LIN {X 0,Y 573.238,Z 329.704,A -85,B 0,C 180,E1 -2317.662,E2 -2317.662} C_VEL
LIN {X 0,Y 573.282,Z 329.698,A -85,B 0,C 180,E1 -2320.728,E2 -2320.728} C_VEL
LIN {X 0,Y 573.255,Z 329.702,A -85,B 0,C 180,E1 -2323.622,E2 -2323.622} C_VEL
LIN {X 0,Y 573.278,Z 329.701,A -85,B 0,C 180,E1 -2325.807,E2 -2325.807} C_VEL
LIN {X 0,Y 573.267,Z 329.702,A -85,B 0,C 180,E1 -2328.745,E2 -2328.745} C_VEL
LIN {X 0,Y 573.287,Z 329.698,A -85,B 0,C 180,E1 -2331.541,E2 -2331.541} C_VEL
LIN {X 0,Y 573.291,Z 329.697,A -85,B 0,C 180,E1 -2334.372,E2 -2334.372} C_VEL
LIN {X 0,Y 573.311,Z 329.696,A -85,B 0,C 180,E1 -2337.893,E2 -2337.893} C_VEL
LIN {X 0,Y 573.336,Z 329.691,A -85,B 0,C 180,E1 -2340.702,E2 -2340.702} C_VEL
LIN {X 0,Y 573.239,Z 329.703,A -85,B 0,C 180,E1 -2343.515,E2 -2343.515} C_VEL
LIN {X 0,Y 573.297,Z 329.699,A -85,B 0,C 180,E1 -2345.628,E2 -2345.628} C_VEL
LIN {X 0,Y 573.292,Z 329.697,A -85,B 0,C 180,E1 -2348.459,E2 -2348.459} C_VEL
LIN {X 0,Y 573.276,Z 329.697,A -85,B 0,C 180,E1 -2351.312,E2 -2351.312} C_VEL
LIN {X 0,Y 573.285,Z 329.696,A -85,B 0,C 180,E1 -2354.424,E2 -2354.424} C_VEL
LIN {X 0,Y 573.264,Z 329.701,A -85,B 0,C 180,E1 -2357.112,E2 -2357.112} C_VEL
LIN {X 0,Y 573.255,Z 329.699,A -85,B 0,C 180,E1 -2360.077,E2 -2360.077} C_VEL
LIN {X 0,Y 573.238,Z 329.704,A -85,B 0,C 180,E1 -2363.099,E2 -2363.099} C_VEL
LIN {X 0,Y 573.252,Z 329.701,A -85,B 0,C 180,E1 -2364.385,E2 -2364.385} C_VEL
LIN {X 0,Y 572.628,Z 329.781,A -85,B 0,C 180,E1 -2364.971,E2 -2364.971} C_VEL
LIN {X 0,Y 569.787,Z 330.139,A -85,B 0,C 180,E1 -2365.922,E2 -2365.922} C_VEL
LIN {X 0,Y 567.354,Z 330.442,A -85,B 0,C 180,E1 -2366.688,E2 -2366.688} C_VEL
LIN {X 0,Y 566.298,Z 330.571,A -85,B 0,C 180,E1 -2367.279,E2 -2367.279} C_VEL
LIN {X 0,Y 566.207,Z 330.58,A -85,B 0,C 180,E1 -2367.479,E2 -2367.479} C_VEL
LIN {X 0,Y 566.205,Z 330.58,A -85,B 0,C 180,E1 -2369.769,E2 -2369.769} C_VEL
LIN {X 0,Y 566.207,Z 330.578,A -85,B 0,C 180,E1 -2372.43,E2 -2372.43} C_VEL
LIN {X 0,Y 566.206,Z 330.584,A -85,B 0,C 180,E1 -2374.993,E2 -2374.993} C_VEL
LIN {X 0,Y 566.2,Z 330.581,A -85,B 0,C 180,E1 -2377.461,E2 -2377.461} C_VEL
LIN {X 0,Y 566.222,Z 330.578,A -85,B 0,C 180,E1 -2380.198,E2 -2380.198} C_VEL
LIN {X 0,Y 566.204,Z 330.58,A -85,B 0,C 180,E1 -2383.054,E2 -2383.054} C_VEL
LIN {X 0,Y 566.202,Z 330.581,A -85,B 0,C 180,E1 -2386.049,E2 -2386.049} C_VEL
LIN {X 0,Y 566.132,Z 330.595,A -85,B 0,C 180,E1 -2388.856,E2 -2388.856} C_VEL
LIN {X 0,Y 566.084,Z 331.003,A -85,B 0,C 180,E1 -2389.79,E2 -2389.79} C_VEL
LIN {X 0,Y 566.074,Z 333.817,A -85,B 0,C 180,E1 -2392.616,E2 -2392.616} C_VEL
LIN {X 0,Y 566.042,Z 336.324,A -85,B 0,C 180,E1 -2395.17,E2 -2395.17} C_VEL
LIN {X 0,Y 566.028,Z 338.882,A -85,B 0,C 180,E1 -2397.73,E2 -2397.73} C_VEL
LIN {X 0,Y 566.001,Z 341.587,A -85,B 0,C 180,E1 -2400.364,E2 -2400.364} C_VEL
LIN {X 0,Y 565.931,Z 344.797,A -85,B 0,C 180,E1 -2403.444,E2 -2403.444} C_VEL
LIN {X 0,Y 565.906,Z 347.412,A -85,B 0,C 180,E1 -2405.806,E2 -2405.806} C_VEL
LIN {X 0,Y 565.904,Z 351.128,A -85,B 0,C 180,E1 -2408.89,E2 -2408.89} C_VEL
LIN {X 0,Y 565.866,Z 354.845,A -85,B 0,C 180,E1 -2411.911,E2 -2411.911} C_VEL
LIN {X 0,Y 565.878,Z 355.244,A -85,B 0,C 180,E1 -2412.232,E2 -2412.232} C_VEL
LIN {X 0,Y 567.937,Z 363.992,A -85,B 0,C 180,E1 -2412.448,E2 -2412.448} C_VEL
LIN {X 0,Y 567.807,Z 378.874,A -85,B 0,C 180,E1 -2412.799,E2 -2412.799} C_VEL
LIN {X 0,Y 567.62,Z 393.572,A -85,B 0,C 180,E1 -2413.29,E2 -2413.29} C_VEL
LIN {X 0,Y 567.404,Z 407.73,A -85,B 0,C 180,E1 -2413.91,E2 -2413.91} C_VEL
LIN {X 0,Y 567.144,Z 421.039,A -85,B 0,C 180,E1 -2414.64,E2 -2414.64} C_VEL
LIN {X 0,Y 566.919,Z 433.971,A -85,B 0,C 180,E1 -2415.507,E2 -2415.507} C_VEL
LIN {X 0,Y 566.651,Z 446.885,A -85,B 0,C 180,E1 -2416.552,E2 -2416.552} C_VEL
LIN {X 0,Y 566.463,Z 458.082,A -85,B 0,C 180,E1 -2417.642,E2 -2417.642} C_VEL
LIN {X 0,Y 566.264,Z 468.177,A -85,B 0,C 180,E1 -2418.809,E2 -2418.809} C_VEL
LIN {X 0,Y 566.133,Z 478.002,A -85,B 0,C 180,E1 -2420.172,E2 -2420.172} C_VEL
LIN {X 0,Y 566.064,Z 485.494,A -85,B 0,C 180,E1 -2421.431,E2 -2421.431} C_VEL
LIN {X 0,Y 565.976,Z 492.498,A -85,B 0,C 180,E1 -2422.867,E2 -2422.867} C_VEL
LIN {X 0,Y 565.982,Z 498.007,A -85,B 0,C 180,E1 -2424.299,E2 -2424.299} C_VEL
LIN {X 0,Y 565.913,Z 502.177,A -85,B 0,C 180,E1 -2425.726,E2 -2425.726} C_VEL
LIN {X 0,Y 565.872,Z 505.114,A -85,B 0,C 180,E1 -2427.152,E2 -2427.152} C_VEL
LIN {X 0,Y 565.842,Z 506.88,A -85,B 0,C 180,E1 -2428.576,E2 -2428.576} C_VEL
LIN {X 0,Y 565.837,Z 507.496,A -85,B 0,C 180,E1 -2430,E2 -2430} C_VEL
LIN {X 0,Y 565.844,Z 506.942,A -85,B 0,C 180,E1 -2431.423,E2 -2431.423} C_VEL
LIN {X 0,Y 565.874,Z 505.259,A -85,B 0,C 180,E1 -2432.847,E2 -2432.847} C_VEL
LIN {X 0,Y 565.913,Z 502.404,A -85,B 0,C 180,E1 -2434.273,E2 -2434.273} C_VEL
LIN {X 0,Y 565.975,Z 498.319,A -85,B 0,C 180,E1 -2435.701,E2 -2435.701} C_VEL
LIN {X 0,Y 565.975,Z 492.905,A -85,B 0,C 180,E1 -2437.133,E2 -2437.133} C_VEL
LIN {X 0,Y 566.061,Z 486.005,A -85,B 0,C 180,E1 -2438.568,E2 -2438.568} C_VEL
LIN {X 0,Y 566.177,Z 477.397,A -85,B 0,C 180,E1 -2440.008,E2 -2440.008} C_VEL
LIN {X 0,Y 566.25,Z 468.953,A -85,B 0,C 180,E1 -2441.183,E2 -2441.183} C_VEL
LIN {X 0,Y 566.436,Z 458.917,A -85,B 0,C 180,E1 -2442.358,E2 -2442.358} C_VEL
LIN {X 0,Y 566.668,Z 446.873,A -85,B 0,C 180,E1 -2443.538,E2 -2443.538} C_VEL
LIN {X 0,Y 566.871,Z 435.302,A -85,B 0,C 180,E1 -2444.484,E2 -2444.484} C_VEL
LIN {X 0,Y 567.148,Z 422.48,A -85,B 0,C 180,E1 -2445.359,E2 -2445.359} C_VEL
LIN {X 0,Y 567.374,Z 409.469,A -85,B 0,C 180,E1 -2446.09,E2 -2446.09} C_VEL
LIN {X 0,Y 567.587,Z 395.421,A -85,B 0,C 180,E1 -2446.725,E2 -2446.725} C_VEL
LIN {X 0,Y 567.79,Z 380.271,A -85,B 0,C 180,E1 -2447.249,E2 -2447.249} C_VEL
LIN {X 0,Y 567.911,Z 365.71,A -85,B 0,C 180,E1 -2447.608,E2 -2447.608} C_VEL
LIN {X 0,Y 567.553,Z 362.338,A -85,B 0,C 180,E1 -2447.688,E2 -2447.688} C_VEL
LIN {X 0,Y 565.868,Z 355.244,A -85,B 0,C 180,E1 -2447.858,E2 -2447.858} C_VEL
LIN {X 0,Y 565.88,Z 352.168,A -85,B 0,C 180,E1 -2450.349,E2 -2450.349} C_VEL
LIN {X 0,Y 565.895,Z 348.449,A -85,B 0,C 180,E1 -2453.416,E2 -2453.416} C_VEL
LIN {X 0,Y 565.942,Z 345.739,A -85,B 0,C 180,E1 -2455.762,E2 -2455.762} C_VEL
LIN {X 0,Y 565.96,Z 343.279,A -85,B 0,C 180,E1 -2458.156,E2 -2458.156} C_VEL
LIN {X 0,Y 566.006,Z 340.226,A -85,B 0,C 180,E1 -2461.045,E2 -2461.045} C_VEL
LIN {X 0,Y 566.049,Z 337.269,A -85,B 0,C 180,E1 -2463.967,E2 -2463.967} C_VEL
LIN {X 0,Y 566.046,Z 334.704,A -85,B 0,C 180,E1 -2466.581,E2 -2466.581} C_VEL
LIN {X 0,Y 566.062,Z 332.025,A -85,B 0,C 180,E1 -2469.286,E2 -2469.286} C_VEL
LIN {X 0,Y 566.078,Z 330.601,A -85,B 0,C 180,E1 -2470.77,E2 -2470.77} C_VEL
LIN {X 0,Y 566.205,Z 330.585,A -85,B 0,C 180,E1 -2473.053,E2 -2473.053} C_VEL
LIN {X 0,Y 566.198,Z 330.586,A -85,B 0,C 180,E1 -2476.048,E2 -2476.048} C_VEL
LIN {X 0,Y 566.208,Z 330.582,A -85,B 0,C 180,E1 -2478.863,E2 -2478.863} C_VEL
LIN {X 0,Y 566.19,Z 330.582,A -85,B 0,C 180,E1 -2481.637,E2 -2481.637} C_VEL
LIN {X 0,Y 566.212,Z 330.579,A -85,B 0,C 180,E1 -2484.311,E2 -2484.311} C_VEL
LIN {X 0,Y 566.219,Z 330.58,A -85,B 0,C 180,E1 -2486.898,E2 -2486.898} C_VEL
LIN {X 0,Y 566.193,Z 330.582,A -85,B 0,C 180,E1 -2489.408,E2 -2489.408} C_VEL
LIN {X 0,Y 566.227,Z 330.575,A -85,B 0,C 180,E1 -2491.858,E2 -2491.858} C_VEL
LIN {X 0,Y 566.225,Z 330.58,A -85,B 0,C 180,E1 -2494.251,E2 -2494.251} C_VEL
LIN {X 0,Y 566.191,Z 330.581,A -85,B 0,C 180,E1 -2496.713,E2 -2496.713} C_VEL
LIN {X 0,Y 566.213,Z 330.575,A -85,B 0,C 180,E1 -2499.663,E2 -2499.663} C_VEL
LIN {X 0,Y 566.203,Z 330.58,A -85,B 0,C 180,E1 -2502.668,E2 -2502.668} C_VEL
LIN {X 0,Y 566.233,Z 330.574,A -85,B 0,C 180,E1 -2505.627,E2 -2505.627} C_VEL
LIN {X 0,Y 566.233,Z 330.575,A -85,B 0,C 180,E1 -2508.675,E2 -2508.675} C_VEL
LIN {X 0,Y 566.233,Z 330.578,A -85,B 0,C 180,E1 -2511.434,E2 -2511.434} C_VEL
LIN {X 0,Y 566.263,Z 330.576,A -85,B 0,C 180,E1 -2514.302,E2 -2514.302} C_VEL
LIN {X 0,Y 566.277,Z 330.571,A -85,B 0,C 180,E1 -2517.866,E2 -2517.866} C_VEL
LIN {X 0,Y 566.303,Z 330.568,A -85,B 0,C 180,E1 -2520.711,E2 -2520.711} C_VEL
LIN {X 0,Y 566.276,Z 330.572,A -85,B 0,C 180,E1 -2522.845,E2 -2522.845} C_VEL
LIN {X 0,Y 566.259,Z 330.573,A -85,B 0,C 180,E1 -2525.698,E2 -2525.698} C_VEL
LIN {X 0,Y 566.228,Z 330.577,A -85,B 0,C 180,E1 -2528.566,E2 -2528.566} C_VEL
LIN {X 0,Y 566.25,Z 330.574,A -85,B 0,C 180,E1 -2531.454,E2 -2531.454} C_VEL
LIN {X 0,Y 566.233,Z 330.576,A -85,B 0,C 180,E1 -2534.507,E2 -2534.507} C_VEL
LIN {X 0,Y 566.199,Z 330.582,A -85,B 0,C 180,E1 -2537.332,E2 -2537.332} C_VEL
LIN {X 0,Y 566.212,Z 330.58,A -85,B 0,C 180,E1 -2540.337,E2 -2540.337} C_VEL
LIN {X 0,Y 566.188,Z 330.584,A -85,B 0,C 180,E1 -2543.404,E2 -2543.404} C_VEL
LIN {X 0,Y 566.212,Z 330.581,A -85,B 0,C 180,E1 -2545.749,E2 -2545.749} C_VEL
LIN {X 0,Y 566.2,Z 330.581,A -85,B 0,C 180,E1 -2548.202,E2 -2548.202} C_VEL
LIN {X 0,Y 566.193,Z 330.586,A -85,B 0,C 180,E1 -2550.592,E2 -2550.592} C_VEL
LIN {X 0,Y 566.227,Z 330.578,A -85,B 0,C 180,E1 -2553.102,E2 -2553.102} C_VEL
LIN {X 0,Y 566.211,Z 330.581,A -85,B 0,C 180,E1 -2555.689,E2 -2555.689} C_VEL
LIN {X 0,Y 566.216,Z 330.581,A -85,B 0,C 180,E1 -2558.559,E2 -2558.559} C_VEL
LIN {X 0,Y 566.211,Z 330.583,A -85,B 0,C 180,E1 -2561.136,E2 -2561.136} C_VEL
LIN {X 0,Y 566.195,Z 330.584,A -85,B 0,C 180,E1 -2564.036,E2 -2564.036} C_VEL
LIN {X 0,Y 566.24,Z 330.749,A -85,B 0,C 180,E1 -2567.079,E2 -2567.079} C_VEL
LIN {X 0,Y 566.797,Z 335.443,A -85,B 0,C 180,E1 -2569.145,E2 -2569.145} C_VEL
LIN {X 0,Y 566.637,Z 342.907,A -85,B 0,C 180,E1 -2572.125,E2 -2572.125} C_VEL
LIN {X 0,Y 566.573,Z 348.853,A -85,B 0,C 180,E1 -2574.338,E2 -2574.338} C_VEL
LIN {X 0,Y 566.495,Z 356.024,A -85,B 0,C 180,E1 -2576.916,E2 -2576.916} C_VEL
LIN {X 0,Y 566.454,Z 363.225,A -85,B 0,C 180,E1 -2579.424,E2 -2579.424} C_VEL
LIN {X 0,Y 566.367,Z 371.685,A -85,B 0,C 180,E1 -2582.269,E2 -2582.269} C_VEL
LIN {X 0,Y 566.318,Z 379.997,A -85,B 0,C 180,E1 -2585.043,E2 -2585.043} C_VEL
LIN {X 0,Y 566.207,Z 389.338,A -85,B 0,C 180,E1 -2588.138,E2 -2588.138} C_VEL
LIN {X 0,Y 566.13,Z 398.678,A -85,B 0,C 180,E1 -2591.17,E2 -2591.17} C_VEL
LIN {X 0,Y 566.103,Z 401.758,A -85,B 0,C 180,E1 -2592.152,E2 -2592.152} C_VEL
LIN {X 0,Y 567.951,Z 409.837,A -85,B 0,C 180,E1 -2592.33,E2 -2592.33} C_VEL
LIN {X 0,Y 567.836,Z 425.005,A -85,B 0,C 180,E1 -2592.65,E2 -2592.65} C_VEL
LIN {X 0,Y 567.714,Z 439.216,A -85,B 0,C 180,E1 -2593.087,E2 -2593.087} C_VEL
LIN {X 0,Y 567.455,Z 452.827,A -85,B 0,C 180,E1 -2593.635,E2 -2593.635} C_VEL
LIN {X 0,Y 567.231,Z 467.106,A -85,B 0,C 180,E1 -2594.367,E2 -2594.367} C_VEL
LIN {X 0,Y 566.972,Z 480.401,A -85,B 0,C 180,E1 -2595.209,E2 -2595.209} C_VEL
LIN {X 0,Y 566.756,Z 493.165,A -85,B 0,C 180,E1 -2596.19,E2 -2596.19} C_VEL
LIN {X 0,Y 566.545,Z 504.973,A -85,B 0,C 180,E1 -2597.28,E2 -2597.28} C_VEL
LIN {X 0,Y 566.343,Z 514.905,A -85,B 0,C 180,E1 -2598.367,E2 -2598.367} C_VEL
LIN {X 0,Y 566.204,Z 524.622,A -85,B 0,C 180,E1 -2599.632,E2 -2599.632} C_VEL
LIN {X 0,Y 566.079,Z 532.724,A -85,B 0,C 180,E1 -2600.892,E2 -2600.892} C_VEL
LIN {X 0,Y 566.014,Z 539.426,A -85,B 0,C 180,E1 -2602.15,E2 -2602.15} C_VEL
LIN {X 0,Y 565.942,Z 545.608,A -85,B 0,C 180,E1 -2603.583,E2 -2603.583} C_VEL
LIN {X 0,Y 565.866,Z 550.386,A -85,B 0,C 180,E1 -2605.013,E2 -2605.013} C_VEL
LIN {X 0,Y 565.909,Z 553.89,A -85,B 0,C 180,E1 -2606.44,E2 -2606.44} C_VEL
LIN {X 0,Y 565.839,Z 556.192,A -85,B 0,C 180,E1 -2607.865,E2 -2607.865} C_VEL
LIN {X 0,Y 565.839,Z 557.349,A -85,B 0,C 180,E1 -2609.289,E2 -2609.289} C_VEL
LIN {X 0,Y 565.839,Z 557.349,A -85,B 0,C 180,E1 -2610.712,E2 -2610.712} C_VEL
LIN {X 0,Y 565.839,Z 556.19,A -85,B 0,C 180,E1 -2612.136,E2 -2612.136} C_VEL
LIN {X 0,Y 565.909,Z 553.886,A -85,B 0,C 180,E1 -2613.56,E2 -2613.56} C_VEL
LIN {X 0,Y 565.867,Z 550.384,A -85,B 0,C 180,E1 -2614.988,E2 -2614.988} C_VEL
LIN {X 0,Y 565.943,Z 545.607,A -85,B 0,C 180,E1 -2616.417,E2 -2616.417} C_VEL
LIN {X 0,Y 566.014,Z 539.421,A -85,B 0,C 180,E1 -2617.85,E2 -2617.85} C_VEL
LIN {X 0,Y 566.071,Z 531.646,A -85,B 0,C 180,E1 -2619.288,E2 -2619.288} C_VEL
LIN {X 0,Y 566.24,Z 523.367,A -85,B 0,C 180,E1 -2620.549,E2 -2620.549} C_VEL
LIN {X 0,Y 566.367,Z 513.389,A -85,B 0,C 180,E1 -2621.815,E2 -2621.815} C_VEL
LIN {X 0,Y 566.586,Z 503.186,A -85,B 0,C 180,E1 -2622.902,E2 -2622.902} C_VEL
LIN {X 0,Y 566.763,Z 491.015,A -85,B 0,C 180,E1 -2623.993,E2 -2623.993} C_VEL
LIN {X 0,Y 567.042,Z 478.336,A -85,B 0,C 180,E1 -2624.936,E2 -2624.936} C_VEL
LIN {X 0,Y 567.267,Z 465.51,A -85,B 0,C 180,E1 -2625.725,E2 -2625.725} C_VEL
LIN {X 0,Y 567.494,Z 450.825,A -85,B 0,C 180,E1 -2626.457,E2 -2626.457} C_VEL
LIN {X 0,Y 567.738,Z 435.318,A -85,B 0,C 180,E1 -2627.051,E2 -2627.051} C_VEL
LIN {X 0,Y 567.923,Z 419.647,A -85,B 0,C 180,E1 -2627.482,E2 -2627.482} C_VEL
LIN {X 0,Y 567.8,Z 409.229,A -85,B 0,C 180,E1 -2627.684,E2 -2627.684} C_VEL
LIN {X 0,Y 566.109,Z 401.681,A -85,B 0,C 180,E1 -2627.867,E2 -2627.867} C_VEL
LIN {X 0,Y 566.183,Z 392.838,A -85,B 0,C 180,E1 -2630.718,E2 -2630.718} C_VEL
LIN {X 0,Y 566.257,Z 383.498,A -85,B 0,C 180,E1 -2633.789,E2 -2633.789} C_VEL
LIN {X 0,Y 566.384,Z 374.811,A -85,B 0,C 180,E1 -2636.695,E2 -2636.695} C_VEL
LIN {X 0,Y 566.417,Z 365.653,A -85,B 0,C 180,E1 -2639.757,E2 -2639.757} C_VEL
LIN {X 0,Y 566.497,Z 357.746,A -85,B 0,C 180,E1 -2642.477,E2 -2642.477} C_VEL
LIN {X 0,Y 566.581,Z 348.832,A -85,B 0,C 180,E1 -2645.662,E2 -2645.662} C_VEL
LIN {X 0,Y 566.664,Z 340.995,A -85,B 0,C 180,E1 -2648.616,E2 -2648.616} C_VEL
LIN {X 0,Y 566.767,Z 334.885,A -85,B 0,C 180,E1 -2651.088,E2 -2651.088} C_VEL
LIN {X 0,Y 566.218,Z 330.582,A -85,B 0,C 180,E1 -2653.053,E2 -2653.053} C_VEL
LIN {X 0,Y 566.2,Z 330.582,A -85,B 0,C 180,E1 -2656.049,E2 -2656.049} C_VEL
LIN {X 0,Y 566.206,Z 330.581,A -85,B 0,C 180,E1 -2659.215,E2 -2659.215} C_VEL
LIN {X 0,Y 566.192,Z 330.587,A -85,B 0,C 180,E1 -2661.637,E2 -2661.637} C_VEL
LIN {X 0,Y 566.215,Z 330.581,A -85,B 0,C 180,E1 -2664.312,E2 -2664.312} C_VEL
LIN {X 0,Y 566.222,Z 330.578,A -85,B 0,C 180,E1 -2666.898,E2 -2666.898} C_VEL
LIN {X 0,Y 566.184,Z 330.588,A -85,B 0,C 180,E1 -2669.408,E2 -2669.408} C_VEL
LIN {X 0,Y 566.214,Z 330.579,A -85,B 0,C 180,E1 -2671.858,E2 -2671.858} C_VEL
LIN {X 0,Y 566.212,Z 330.581,A -85,B 0,C 180,E1 -2674.251,E2 -2674.251} C_VEL
LIN {X 0,Y 566.172,Z 330.587,A -85,B 0,C 180,E1 -2676.719,E2 -2676.719} C_VEL
LIN {X 0,Y 566.216,Z 330.58,A -85,B 0,C 180,E1 -2679.663,E2 -2679.663} C_VEL
LIN {X 0,Y 566.203,Z 330.582,A -85,B 0,C 180,E1 -2682.669,E2 -2682.669} C_VEL
LIN {X 0,Y 566.238,Z 330.577,A -85,B 0,C 180,E1 -2685.627,E2 -2685.627} C_VEL
LIN {X 0,Y 566.238,Z 330.577,A -85,B 0,C 180,E1 -2688.675,E2 -2688.675} C_VEL
LIN {X 0,Y 566.231,Z 330.577,A -85,B 0,C 180,E1 -2691.434,E2 -2691.434} C_VEL
LIN {X 0,Y 566.26,Z 330.573,A -85,B 0,C 180,E1 -2694.302,E2 -2694.302} C_VEL
LIN {X 0,Y 566.282,Z 330.571,A -85,B 0,C 180,E1 -2697.866,E2 -2697.866} C_VEL
LIN {X 0,Y 566.306,Z 330.567,A -85,B 0,C 180,E1 -2700.711,E2 -2700.711} C_VEL
LIN {X 0,Y 566.28,Z 330.576,A -85,B 0,C 180,E1 -2702.846,E2 -2702.846} C_VEL
LIN {X 0,Y 566.265,Z 330.575,A -85,B 0,C 180,E1 -2705.698,E2 -2705.698} C_VEL
LIN {X 0,Y 566.237,Z 330.577,A -85,B 0,C 180,E1 -2708.566,E2 -2708.566} C_VEL
LIN {X 0,Y 566.246,Z 330.573,A -85,B 0,C 180,E1 -2711.454,E2 -2711.454} C_VEL
LIN {X 0,Y 566.238,Z 330.574,A -85,B 0,C 180,E1 -2714.506,E2 -2714.506} C_VEL
LIN {X 0,Y 566.207,Z 330.579,A -85,B 0,C 180,E1 -2717.331,E2 -2717.331} C_VEL
LIN {X 0,Y 566.216,Z 330.574,A -85,B 0,C 180,E1 -2720.337,E2 -2720.337} C_VEL
LIN {X 0,Y 566.173,Z 330.584,A -85,B 0,C 180,E1 -2723.281,E2 -2723.281} C_VEL
LIN {X 0,Y 566.219,Z 330.581,A -85,B 0,C 180,E1 -2725.749,E2 -2725.749} C_VEL
LIN {X 0,Y 566.207,Z 330.58,A -85,B 0,C 180,E1 -2727.479,E2 -2727.479} C_VEL
LIN {X 0,Y 565.526,Z 330.662,A -85,B 0,C 180,E1 -2728.073,E2 -2728.073} C_VEL
LIN {X 0,Y 562.661,Z 331.023,A -85,B 0,C 180,E1 -2729.037,E2 -2729.037} C_VEL
LIN {X 0,Y 560.252,Z 331.324,A -85,B 0,C 180,E1 -2729.812,E2 -2729.812} C_VEL
LIN {X 0,Y 559.225,Z 331.453,A -85,B 0,C 180,E1 -2730.411,E2 -2730.411} C_VEL
LIN {X 0,Y 559.145,Z 331.459,A -85,B 0,C 180,E1 -2730.614,E2 -2730.614} C_VEL
LIN {X 0,Y 559.166,Z 331.457,A -85,B 0,C 180,E1 -2733.575,E2 -2733.575} C_VEL
LIN {X 0,Y 559.186,Z 331.459,A -85,B 0,C 180,E1 -2736.45,E2 -2736.45} C_VEL
LIN {X 0,Y 559.182,Z 331.455,A -85,B 0,C 180,E1 -2738.934,E2 -2738.934} C_VEL
LIN {X 0,Y 559.169,Z 331.456,A -85,B 0,C 180,E1 -2741.77,E2 -2741.77} C_VEL
LIN {X 0,Y 559.143,Z 331.46,A -85,B 0,C 180,E1 -2744.739,E2 -2744.739} C_VEL
LIN {X 0,Y 559.161,Z 331.461,A -85,B 0,C 180,E1 -2747.256,E2 -2747.256} C_VEL
LIN {X 0,Y 559.047,Z 331.477,A -85,B 0,C 180,E1 -2749.178,E2 -2749.178} C_VEL
LIN {X 0,Y 559.021,Z 332.987,A -85,B 0,C 180,E1 -2751.053,E2 -2751.053} C_VEL
LIN {X 0,Y 559.001,Z 335.638,A -85,B 0,C 180,E1 -2753.778,E2 -2753.778} C_VEL
LIN {X 0,Y 558.986,Z 338.223,A -85,B 0,C 180,E1 -2756.413,E2 -2756.413} C_VEL
LIN {X 0,Y 558.95,Z 340.791,A -85,B 0,C 180,E1 -2758.968,E2 -2758.968} C_VEL
LIN {X 0,Y 558.88,Z 343.567,A -85,B 0,C 180,E1 -2761.674,E2 -2761.674} C_VEL
LIN {X 0,Y 558.84,Z 346.724,A -85,B 0,C 180,E1 -2764.685,E2 -2764.685} C_VEL
LIN {X 0,Y 558.795,Z 349.271,A -85,B 0,C 180,E1 -2767.052,E2 -2767.052} C_VEL
LIN {X 0,Y 558.786,Z 352.058,A -85,B 0,C 180,E1 -2769.38,E2 -2769.38} C_VEL
LIN {X 0,Y 558.803,Z 355.233,A -85,B 0,C 180,E1 -2771.989,E2 -2771.989} C_VEL
LIN {X 0,Y 561.17,Z 365.212,A -85,B 0,C 180,E1 -2772.254,E2 -2772.254} C_VEL
LIN {X 0,Y 560.999,Z 380.473,A -85,B 0,C 180,E1 -2772.632,E2 -2772.632} C_VEL
LIN {X 0,Y 560.746,Z 395.731,A -85,B 0,C 180,E1 -2773.168,E2 -2773.168} C_VEL
LIN {X 0,Y 560.52,Z 409.505,A -85,B 0,C 180,E1 -2773.8,E2 -2773.8} C_VEL
LIN {X 0,Y 560.232,Z 422.508,A -85,B 0,C 180,E1 -2774.539,E2 -2774.539} C_VEL
LIN {X 0,Y 559.958,Z 435.79,A -85,B 0,C 180,E1 -2775.462,E2 -2775.462} C_VEL
LIN {X 0,Y 559.691,Z 446.892,A -85,B 0,C 180,E1 -2776.382,E2 -2776.382} C_VEL
LIN {X 0,Y 559.487,Z 458.087,A -85,B 0,C 180,E1 -2777.485,E2 -2777.485} C_VEL
LIN {X 0,Y 559.229,Z 468.785,A -85,B 0,C 180,E1 -2778.743,E2 -2778.743} C_VEL
LIN {X 0,Y 559.096,Z 478.006,A -85,B 0,C 180,E1 -2780.047,E2 -2780.047} C_VEL
LIN {X 0,Y 559.002,Z 485.496,A -85,B 0,C 180,E1 -2781.322,E2 -2781.322} C_VEL
LIN {X 0,Y 558.901,Z 492.5,A -85,B 0,C 180,E1 -2782.776,E2 -2782.776} C_VEL
LIN {X 0,Y 558.888,Z 498.009,A -85,B 0,C 180,E1 -2784.226,E2 -2784.226} C_VEL
LIN {X 0,Y 558.808,Z 502.178,A -85,B 0,C 180,E1 -2785.672,E2 -2785.672} C_VEL
LIN {X 0,Y 558.793,Z 505.114,A -85,B 0,C 180,E1 -2787.116,E2 -2787.116} C_VEL
LIN {X 0,Y 558.742,Z 506.879,A -85,B 0,C 180,E1 -2788.558,E2 -2788.558} C_VEL
LIN {X 0,Y 558.738,Z 507.496,A -85,B 0,C 180,E1 -2790,E2 -2790} C_VEL
LIN {X 0,Y 558.744,Z 506.941,A -85,B 0,C 180,E1 -2791.441,E2 -2791.441} C_VEL
LIN {X 0,Y 558.795,Z 505.257,A -85,B 0,C 180,E1 -2792.883,E2 -2792.883} C_VEL
LIN {X 0,Y 558.808,Z 502.403,A -85,B 0,C 180,E1 -2794.327,E2 -2794.327} C_VEL
LIN {X 0,Y 558.881,Z 498.317,A -85,B 0,C 180,E1 -2795.773,E2 -2795.773} C_VEL
LIN {X 0,Y 558.9,Z 492.902,A -85,B 0,C 180,E1 -2797.224,E2 -2797.224} C_VEL
LIN {X 0,Y 559.001,Z 486.001,A -85,B 0,C 180,E1 -2798.677,E2 -2798.677} C_VEL
LIN {X 0,Y 559.091,Z 478.573,A -85,B 0,C 180,E1 -2799.953,E2 -2799.953} C_VEL
LIN {X 0,Y 559.215,Z 469.511,A -85,B 0,C 180,E1 -2801.25,E2 -2801.25} C_VEL
LIN {X 0,Y 559.451,Z 458.912,A -85,B 0,C 180,E1 -2802.515,E2 -2802.515} C_VEL
LIN {X 0,Y 559.696,Z 446.867,A -85,B 0,C 180,E1 -2803.71,E2 -2803.71} C_VEL
LIN {X 0,Y 559.959,Z 434.395,A -85,B 0,C 180,E1 -2804.736,E2 -2804.736} C_VEL
LIN {X 0,Y 560.261,Z 421.008,A -85,B 0,C 180,E1 -2805.646,E2 -2805.646} C_VEL
LIN {X 0,Y 560.544,Z 407.689,A -85,B 0,C 180,E1 -2806.385,E2 -2806.385} C_VEL
LIN {X 0,Y 560.839,Z 392.535,A -85,B 0,C 180,E1 -2807.051,E2 -2807.051} C_VEL
LIN {X 0,Y 561.074,Z 377.642,A -85,B 0,C 180,E1 -2807.542,E2 -2807.542} C_VEL
LIN {X 0,Y 561.021,Z 364.523,A -85,B 0,C 180,E1 -2807.855,E2 -2807.855} C_VEL
LIN {X 0,Y 558.776,Z 355.231,A -85,B 0,C 180,E1 -2808.102,E2 -2808.102} C_VEL
LIN {X 0,Y 558.785,Z 352.168,A -85,B 0,C 180,E1 -2810.619,E2 -2810.619} C_VEL
LIN {X 0,Y 558.827,Z 348.894,A -85,B 0,C 180,E1 -2813.354,E2 -2813.354} C_VEL
LIN {X 0,Y 558.861,Z 345.991,A -85,B 0,C 180,E1 -2816.113,E2 -2816.113} C_VEL
LIN {X 0,Y 558.875,Z 343.471,A -85,B 0,C 180,E1 -2818.545,E2 -2818.545} C_VEL
LIN {X 0,Y 558.931,Z 340.676,A -85,B 0,C 180,E1 -2821.237,E2 -2821.237} C_VEL
LIN {X 0,Y 558.992,Z 337.977,A -85,B 0,C 180,E1 -2823.922,E2 -2823.922} C_VEL
LIN {X 0,Y 559.001,Z 335.541,A -85,B 0,C 180,E1 -2826.425,E2 -2826.425} C_VEL
LIN {X 0,Y 559.026,Z 333.083,A -85,B 0,C 180,E1 -2828.946,E2 -2828.946} C_VEL
LIN {X 0,Y 559.039,Z 331.478,A -85,B 0,C 180,E1 -2830.822,E2 -2830.822} C_VEL
LIN {X 0,Y 559.168,Z 331.46,A -85,B 0,C 180,E1 -2833.199,E2 -2833.199} C_VEL
LIN {X 0,Y 559.141,Z 331.463,A -85,B 0,C 180,E1 -2836.266,E2 -2836.266} C_VEL
LIN {X 0,Y 559.175,Z 331.461,A -85,B 0,C 180,E1 -2839.189,E2 -2839.189} C_VEL
LIN {X 0,Y 559.135,Z 331.464,A -85,B 0,C 180,E1 -2841.982,E2 -2841.982} C_VEL
LIN {X 0,Y 559.158,Z 331.458,A -85,B 0,C 180,E1 -2844.678,E2 -2844.678} C_VEL
LIN {X 0,Y 559.155,Z 331.456,A -85,B 0,C 180,E1 -2847.364,E2 -2847.364} C_VEL
LIN {X 0,Y 559.188,Z 331.455,A -85,B 0,C 180,E1 -2850.135,E2 -2850.135} C_VEL
LIN {X 0,Y 559.182,Z 331.454,A -85,B 0,C 180,E1 -2853.17,E2 -2853.17} C_VEL
LIN {X 0,Y 559.156,Z 331.459,A -85,B 0,C 180,E1 -2855.495,E2 -2855.495} C_VEL
LIN {X 0,Y 559.17,Z 331.456,A -85,B 0,C 180,E1 -2858.624,E2 -2858.624} C_VEL
LIN {X 0,Y 559.17,Z 331.455,A -85,B 0,C 180,E1 -2860.926,E2 -2860.926} C_VEL
LIN {X 0,Y 559.17,Z 331.456,A -85,B 0,C 180,E1 -2863.948,E2 -2863.948} C_VEL
LIN {X 0,Y 559.173,Z 331.455,A -85,B 0,C 180,E1 -2866.184,E2 -2866.184} C_VEL
LIN {X 0,Y 559.204,Z 331.451,A -85,B 0,C 180,E1 -2868.604,E2 -2868.604} C_VEL
LIN {X 0,Y 559.192,Z 331.456,A -85,B 0,C 180,E1 -2871.326,E2 -2871.326} C_VEL
LIN {X 0,Y 559.232,Z 331.453,A -85,B 0,C 180,E1 -2874.23,E2 -2874.23} C_VEL
LIN {X 0,Y 559.249,Z 331.446,A -85,B 0,C 180,E1 -2877.839,E2 -2877.839} C_VEL
LIN {X 0,Y 559.273,Z 331.444,A -85,B 0,C 180,E1 -2880.72,E2 -2880.72} C_VEL
LIN {X 0,Y 559.242,Z 331.448,A -85,B 0,C 180,E1 -2882.881,E2 -2882.881} C_VEL
LIN {X 0,Y 559.228,Z 331.449,A -85,B 0,C 180,E1 -2885.77,E2 -2885.77} C_VEL
LIN {X 0,Y 559.186,Z 331.454,A -85,B 0,C 180,E1 -2888.674,E2 -2888.674} C_VEL
LIN {X 0,Y 559.208,Z 331.451,A -85,B 0,C 180,E1 -2891.6,E2 -2891.6} C_VEL
LIN {X 0,Y 559.198,Z 331.452,A -85,B 0,C 180,E1 -2894.596,E2 -2894.596} C_VEL
LIN {X 0,Y 559.158,Z 331.457,A -85,B 0,C 180,E1 -2897.557,E2 -2897.557} C_VEL
LIN {X 0,Y 559.17,Z 331.46,A -85,B 0,C 180,E1 -2899.837,E2 -2899.837} C_VEL
LIN {X 0,Y 559.141,Z 331.46,A -85,B 0,C 180,E1 -2902.153,E2 -2902.153} C_VEL
LIN {X 0,Y 559.177,Z 331.456,A -85,B 0,C 180,E1 -2905.187,E2 -2905.187} C_VEL
LIN {X 0,Y 559.188,Z 331.459,A -85,B 0,C 180,E1 -2907.712,E2 -2907.712} C_VEL
LIN {X 0,Y 559.167,Z 331.458,A -85,B 0,C 180,E1 -2910.182,E2 -2910.182} C_VEL
LIN {X 0,Y 559.173,Z 331.457,A -85,B 0,C 180,E1 -2912.714,E2 -2912.714} C_VEL
LIN {X 0,Y 559.157,Z 331.463,A -85,B 0,C 180,E1 -2915.322,E2 -2915.322} C_VEL
LIN {X 0,Y 559.135,Z 331.464,A -85,B 0,C 180,E1 -2918.017,E2 -2918.017} C_VEL
LIN {X 0,Y 559.175,Z 331.457,A -85,B 0,C 180,E1 -2920.811,E2 -2920.811} C_VEL
LIN {X 0,Y 559.139,Z 331.462,A -85,B 0,C 180,E1 -2923.734,E2 -2923.734} C_VEL
LIN {X 0,Y 559.193,Z 331.589,A -85,B 0,C 180,E1 -2926.798,E2 -2926.798} C_VEL
LIN {X 0,Y 559.825,Z 336.206,A -85,B 0,C 180,E1 -2928.871,E2 -2928.871} C_VEL
LIN {X 0,Y 559.686,Z 342.815,A -85,B 0,C 180,E1 -2931.575,E2 -2931.575} C_VEL
LIN {X 0,Y 559.588,Z 349.894,A -85,B 0,C 180,E1 -2934.268,E2 -2934.268} C_VEL
LIN {X 0,Y 559.493,Z 357.051,A -85,B 0,C 180,E1 -2936.879,E2 -2936.879} C_VEL
LIN {X 0,Y 559.421,Z 364.245,A -85,B 0,C 180,E1 -2939.416,E2 -2939.416} C_VEL
LIN {X 0,Y 559.329,Z 371.632,A -85,B 0,C 180,E1 -2941.94,E2 -2941.94} C_VEL
LIN {X 0,Y 559.301,Z 379.93,A -85,B 0,C 180,E1 -2944.708,E2 -2944.708} C_VEL
LIN {X 0,Y 559.164,Z 389.338,A -85,B 0,C 180,E1 -2947.849,E2 -2947.849} C_VEL
LIN {X 0,Y 559.096,Z 397.448,A -85,B 0,C 180,E1 -2950.522,E2 -2950.522} C_VEL
LIN {X 0,Y 559.035,Z 401.72,A -85,B 0,C 180,E1 -2951.912,E2 -2951.912} C_VEL
LIN {X 0,Y 561.214,Z 411.791,A -85,B 0,C 180,E1 -2952.141,E2 -2952.141} C_VEL
LIN {X 0,Y 561.04,Z 427.716,A -85,B 0,C 180,E1 -2952.504,E2 -2952.504} C_VEL
LIN {X 0,Y 560.829,Z 443.375,A -85,B 0,C 180,E1 -2953.028,E2 -2953.028} C_VEL
LIN {X 0,Y 560.563,Z 456.78,A -85,B 0,C 180,E1 -2953.615,E2 -2953.615} C_VEL
LIN {X 0,Y 560.301,Z 470.252,A -85,B 0,C 180,E1 -2954.355,E2 -2954.355} C_VEL
LIN {X 0,Y 560.011,Z 483.473,A -85,B 0,C 180,E1 -2955.243,E2 -2955.243} C_VEL
LIN {X 0,Y 559.702,Z 496.354,A -85,B 0,C 180,E1 -2956.29,E2 -2956.29} C_VEL
LIN {X 0,Y 559.474,Z 508.512,A -85,B 0,C 180,E1 -2957.486,E2 -2957.486} C_VEL
LIN {X 0,Y 559.197,Z 519.243,A -85,B 0,C 180,E1 -2958.758,E2 -2958.758} C_VEL
LIN {X 0,Y 559.091,Z 528.296,A -85,B 0,C 180,E1 -2960.047,E2 -2960.047} C_VEL
LIN {X 0,Y 559,Z 535.752,A -85,B 0,C 180,E1 -2961.323,E2 -2961.323} C_VEL
LIN {X 0,Y 558.899,Z 542.703,A -85,B 0,C 180,E1 -2962.776,E2 -2962.776} C_VEL
LIN {X 0,Y 558.888,Z 548.163,A -85,B 0,C 180,E1 -2964.227,E2 -2964.227} C_VEL
LIN {X 0,Y 558.807,Z 552.292,A -85,B 0,C 180,E1 -2965.673,E2 -2965.673} C_VEL
LIN {X 0,Y 558.794,Z 555.187,A -85,B 0,C 180,E1 -2967.117,E2 -2967.117} C_VEL
LIN {X 0,Y 558.743,Z 556.911,A -85,B 0,C 180,E1 -2968.559,E2 -2968.559} C_VEL
LIN {X 0,Y 558.737,Z 557.5,A -85,B 0,C 180,E1 -2970,E2 -2970} C_VEL
LIN {X 0,Y 558.743,Z 556.909,A -85,B 0,C 180,E1 -2971.442,E2 -2971.442} C_VEL
LIN {X 0,Y 558.794,Z 555.184,A -85,B 0,C 180,E1 -2972.884,E2 -2972.884} C_VEL
LIN {X 0,Y 558.807,Z 552.289,A -85,B 0,C 180,E1 -2974.328,E2 -2974.328} C_VEL
LIN {X 0,Y 558.888,Z 548.163,A -85,B 0,C 180,E1 -2975.774,E2 -2975.774} C_VEL
LIN {X 0,Y 558.9,Z 542.7,A -85,B 0,C 180,E1 -2977.224,E2 -2977.224} C_VEL
LIN {X 0,Y 559.001,Z 535.745,A -85,B 0,C 180,E1 -2978.678,E2 -2978.678} C_VEL
LIN {X 0,Y 559.092,Z 528.29,A -85,B 0,C 180,E1 -2979.953,E2 -2979.953} C_VEL
LIN {X 0,Y 559.228,Z 519.119,A -85,B 0,C 180,E1 -2981.258,E2 -2981.258} C_VEL
LIN {X 0,Y 559.475,Z 508.505,A -85,B 0,C 180,E1 -2982.515,E2 -2982.515} C_VEL
LIN {X 0,Y 559.693,Z 496.35,A -85,B 0,C 180,E1 -2983.71,E2 -2983.71} C_VEL
LIN {X 0,Y 560.004,Z 483.519,A -85,B 0,C 180,E1 -2984.754,E2 -2984.754} C_VEL
LIN {X 0,Y 560.302,Z 470.24,A -85,B 0,C 180,E1 -2985.645,E2 -2985.645} C_VEL
LIN {X 0,Y 560.563,Z 456.761,A -85,B 0,C 180,E1 -2986.385,E2 -2986.385} C_VEL
LIN {X 0,Y 560.834,Z 442.225,A -85,B 0,C 180,E1 -2987.018,E2 -2987.018} C_VEL
LIN {X 0,Y 561.078,Z 426.836,A -85,B 0,C 180,E1 -2987.519,E2 -2987.519} C_VEL
LIN {X 0,Y 561.197,Z 411.216,A -85,B 0,C 180,E1 -2987.868,E2 -2987.868} C_VEL
LIN {X 0,Y 559.045,Z 401.693,A -85,B 0,C 180,E1 -2988.097,E2 -2988.097} C_VEL
LIN {X 0,Y 559.144,Z 392.838,A -85,B 0,C 180,E1 -2990.991,E2 -2990.991} C_VEL
LIN {X 0,Y 559.219,Z 383.498,A -85,B 0,C 180,E1 -2994.107,E2 -2994.107} C_VEL
LIN {X 0,Y 559.338,Z 375.085,A -85,B 0,C 180,E1 -2996.894,E2 -2996.894} C_VEL
LIN {X 0,Y 559.4,Z 366.218,A -85,B 0,C 180,E1 -2999.902,E2 -2999.902} C_VEL
LIN {X 0,Y 559.491,Z 358.249,A -85,B 0,C 180,E1 -3002.694,E2 -3002.694} C_VEL
LIN {X 0,Y 559.594,Z 349.864,A -85,B 0,C 180,E1 -3005.733,E2 -3005.733} C_VEL
LIN {X 0,Y 559.685,Z 342.819,A -85,B 0,C 180,E1 -3008.423,E2 -3008.423} C_VEL
LIN {X 0,Y 559.817,Z 336.2,A -85,B 0,C 180,E1 -3011.128,E2 -3011.128} C_VEL
LIN {X 0,Y 559.166,Z 331.461,A -85,B 0,C 180,E1 -3013.288,E2 -3013.288} C_VEL
LIN {X 0,Y 559.143,Z 331.46,A -85,B 0,C 180,E1 -3016.266,E2 -3016.266} C_VEL
LIN {X 0,Y 559.158,Z 331.459,A -85,B 0,C 180,E1 -3019.188,E2 -3019.188} C_VEL
LIN {X 0,Y 559.138,Z 331.464,A -85,B 0,C 180,E1 -3021.983,E2 -3021.983} C_VEL
LIN {X 0,Y 559.162,Z 331.463,A -85,B 0,C 180,E1 -3024.783,E2 -3024.783} C_VEL
LIN {X 0,Y 559.158,Z 331.459,A -85,B 0,C 180,E1 -3027.365,E2 -3027.365} C_VEL
LIN {X 0,Y 559.151,Z 331.459,A -85,B 0,C 180,E1 -3030.143,E2 -3030.143} C_VEL
LIN {X 0,Y 559.172,Z 331.456,A -85,B 0,C 180,E1 -3033.098,E2 -3033.098} C_VEL
LIN {X 0,Y 559.159,Z 331.463,A -85,B 0,C 180,E1 -3035.495,E2 -3035.495} C_VEL
LIN {X 0,Y 559.175,Z 331.46,A -85,B 0,C 180,E1 -3038.624,E2 -3038.624} C_VEL
LIN {X 0,Y 559.17,Z 331.456,A -85,B 0,C 180,E1 -3040.926,E2 -3040.926} C_VEL
LIN {X 0,Y 559.17,Z 331.457,A -85,B 0,C 180,E1 -3043.948,E2 -3043.948} C_VEL
LIN {X 0,Y 559.177,Z 331.461,A -85,B 0,C 180,E1 -3046.184,E2 -3046.184} C_VEL
LIN {X 0,Y 559.198,Z 331.459,A -85,B 0,C 180,E1 -3049.134,E2 -3049.134} C_VEL
LIN {X 0,Y 559.208,Z 331.456,A -85,B 0,C 180,E1 -3052.054,E2 -3052.054} C_VEL
LIN {X 0,Y 559.258,Z 331.447,A -85,B 0,C 180,E1 -3054.953,E2 -3054.953} C_VEL
LIN {X 0,Y 559.254,Z 331.446,A -85,B 0,C 180,E1 -3057.84,E2 -3057.84} C_VEL
LIN {X 0,Y 559.276,Z 331.443,A -85,B 0,C 180,E1 -3060.72,E2 -3060.72} C_VEL
LIN {X 0,Y 559.246,Z 331.451,A -85,B 0,C 180,E1 -3062.881,E2 -3062.881} C_VEL
LIN {X 0,Y 559.235,Z 331.452,A -85,B 0,C 180,E1 -3065.77,E2 -3065.77} C_VEL
LIN {X 0,Y 559.195,Z 331.455,A -85,B 0,C 180,E1 -3068.674,E2 -3068.674} C_VEL
LIN {X 0,Y 559.21,Z 331.45,A -85,B 0,C 180,E1 -3071.6,E2 -3071.6} C_VEL
LIN {X 0,Y 559.204,Z 331.45,A -85,B 0,C 180,E1 -3074.596,E2 -3074.596} C_VEL
LIN {X 0,Y 559.166,Z 331.457,A -85,B 0,C 180,E1 -3077.557,E2 -3077.557} C_VEL
LIN {X 0,Y 559.173,Z 331.454,A -85,B 0,C 180,E1 -3079.837,E2 -3079.837} C_VEL
LIN {X 0,Y 559.144,Z 331.458,A -85,B 0,C 180,E1 -3082.153,E2 -3082.153} C_VEL
LIN {X 0,Y 559.18,Z 331.455,A -85,B 0,C 180,E1 -3085.298,E2 -3085.298} C_VEL
LIN {X 0,Y 559.161,Z 331.455,A -85,B 0,C 180,E1 -3087.713,E2 -3087.713} C_VEL
LIN {X 0,Y 559.145,Z 331.459,A -85,B 0,C 180,E1 -3090.614,E2 -3090.614} C_VEL
LIN {X 0,Y 558.484,Z 331.542,A -85,B 0,C 180,E1 -3091.215,E2 -3091.215} C_VEL
LIN {X 0,Y 555.62,Z 331.898,A -85,B 0,C 180,E1 -3092.191,E2 -3092.191} C_VEL
LIN {X 0,Y 553.207,Z 332.199,A -85,B 0,C 180,E1 -3092.977,E2 -3092.977} C_VEL
LIN {X 0,Y 552.188,Z 332.326,A -85,B 0,C 180,E1 -3093.583,E2 -3093.583} C_VEL
LIN {X 0,Y 552.114,Z 332.332,A -85,B 0,C 180,E1 -3093.789,E2 -3093.789} C_VEL
LIN {X 0,Y 552.119,Z 332.336,A -85,B 0,C 180,E1 -3096.746,E2 -3096.746} C_VEL
LIN {X 0,Y 552.136,Z 332.337,A -85,B 0,C 180,E1 -3099.527,E2 -3099.527} C_VEL
LIN {X 0,Y 552.133,Z 332.338,A -85,B 0,C 180,E1 -3102.425,E2 -3102.425} C_VEL
LIN {X 0,Y 552.102,Z 332.343,A -85,B 0,C 180,E1 -3105.563,E2 -3105.563} C_VEL
LIN {X 0,Y 552.132,Z 332.334,A -85,B 0,C 180,E1 -3107.585,E2 -3107.585} C_VEL
LIN {X 0,Y 551.954,Z 332.492,A -85,B 0,C 180,E1 -3109.816,E2 -3109.816} C_VEL
LIN {X 0,Y 551.954,Z 334.913,A -85,B 0,C 180,E1 -3112.325,E2 -3112.325} C_VEL
LIN {X 0,Y 551.911,Z 337.549,A -85,B 0,C 180,E1 -3115.038,E2 -3115.038} C_VEL
LIN {X 0,Y 551.874,Z 340.126,A -85,B 0,C 180,E1 -3117.665,E2 -3117.665} C_VEL
LIN {X 0,Y 551.867,Z 342.706,A -85,B 0,C 180,E1 -3120.22,E2 -3120.22} C_VEL
LIN {X 0,Y 551.81,Z 345.621,A -85,B 0,C 180,E1 -3123.067,E2 -3123.067} C_VEL
LIN {X 0,Y 551.73,Z 348.636,A -85,B 0,C 180,E1 -3125.944,E2 -3125.944} C_VEL
LIN {X 0,Y 551.726,Z 351.245,A -85,B 0,C 180,E1 -3128.418,E2 -3128.418} C_VEL
LIN {X 0,Y 551.67,Z 354.847,A -85,B 0,C 180,E1 -3131.428,E2 -3131.428} C_VEL
LIN {X 0,Y 551.698,Z 355.378,A -85,B 0,C 180,E1 -3131.765,E2 -3131.765} C_VEL
LIN {X 0,Y 554.394,Z 367.065,A -85,B 0,C 180,E1 -3132.068,E2 -3132.068} C_VEL
LIN {X 0,Y 554.192,Z 381.933,A -85,B 0,C 180,E1 -3132.457,E2 -3132.457} C_VEL
LIN {X 0,Y 553.949,Z 395.877,A -85,B 0,C 180,E1 -3132.961,E2 -3132.961} C_VEL
LIN {X 0,Y 553.671,Z 409.514,A -85,B 0,C 180,E1 -3133.594,E2 -3133.594} C_VEL
LIN {X 0,Y 553.337,Z 422.515,A -85,B 0,C 180,E1 -3134.341,E2 -3134.341} C_VEL
LIN {X 0,Y 553.038,Z 435.796,A -85,B 0,C 180,E1 -3135.276,E2 -3135.276} C_VEL
LIN {X 0,Y 552.724,Z 446.899,A -85,B 0,C 180,E1 -3136.207,E2 -3136.207} C_VEL
LIN {X 0,Y 552.489,Z 458.093,A -85,B 0,C 180,E1 -3137.324,E2 -3137.324} C_VEL
LIN {X 0,Y 552.199,Z 469.338,A -85,B 0,C 180,E1 -3138.672,E2 -3138.672} C_VEL
LIN {X 0,Y 552.076,Z 478.009,A -85,B 0,C 180,E1 -3139.919,E2 -3139.919} C_VEL
LIN {X 0,Y 551.92,Z 485.499,A -85,B 0,C 180,E1 -3141.21,E2 -3141.21} C_VEL
LIN {X 0,Y 551.821,Z 492.503,A -85,B 0,C 180,E1 -3142.683,E2 -3142.683} C_VEL
LIN {X 0,Y 551.794,Z 498.012,A -85,B 0,C 180,E1 -3144.152,E2 -3144.152} C_VEL
LIN {X 0,Y 551.706,Z 502.179,A -85,B 0,C 180,E1 -3145.616,E2 -3145.616} C_VEL
LIN {X 0,Y 551.717,Z 505.113,A -85,B 0,C 180,E1 -3147.079,E2 -3147.079} C_VEL
LIN {X 0,Y 551.642,Z 506.879,A -85,B 0,C 180,E1 -3148.54,E2 -3148.54} C_VEL
LIN {X 0,Y 551.638,Z 507.496,A -85,B 0,C 180,E1 -3150,E2 -3150} C_VEL
LIN {X 0,Y 551.644,Z 506.94,A -85,B 0,C 180,E1 -3151.46,E2 -3151.46} C_VEL
LIN {X 0,Y 551.719,Z 505.256,A -85,B 0,C 180,E1 -3152.92,E2 -3152.92} C_VEL
LIN {X 0,Y 551.706,Z 502.402,A -85,B 0,C 180,E1 -3154.383,E2 -3154.383} C_VEL
LIN {X 0,Y 551.787,Z 498.315,A -85,B 0,C 180,E1 -3155.848,E2 -3155.848} C_VEL
LIN {X 0,Y 551.82,Z 492.9,A -85,B 0,C 180,E1 -3157.317,E2 -3157.317} C_VEL
LIN {X 0,Y 551.919,Z 485.998,A -85,B 0,C 180,E1 -3158.789,E2 -3158.789} C_VEL
LIN {X 0,Y 552.071,Z 478.57,A -85,B 0,C 180,E1 -3160.081,E2 -3160.081} C_VEL
LIN {X 0,Y 552.183,Z 470.06,A -85,B 0,C 180,E1 -3161.32,E2 -3161.32} C_VEL
LIN {X 0,Y 552.403,Z 460.533,A -85,B 0,C 180,E1 -3162.491,E2 -3162.491} C_VEL
LIN {X 0,Y 552.672,Z 449.802,A -85,B 0,C 180,E1 -3163.606,E2 -3163.606} C_VEL
LIN {X 0,Y 552.95,Z 438.092,A -85,B 0,C 180,E1 -3164.632,E2 -3164.632} C_VEL
LIN {X 0,Y 553.295,Z 425.307,A -85,B 0,C 180,E1 -3165.565,E2 -3165.565} C_VEL
LIN {X 0,Y 553.587,Z 412.97,A -85,B 0,C 180,E1 -3166.313,E2 -3166.313} C_VEL
LIN {X 0,Y 553.868,Z 399.75,A -85,B 0,C 180,E1 -3166.968,E2 -3166.968} C_VEL
LIN {X 0,Y 554.166,Z 385.702,A -85,B 0,C 180,E1 -3167.512,E2 -3167.512} C_VEL
LIN {X 0,Y 554.419,Z 370.137,A -85,B 0,C 180,E1 -3167.955,E2 -3167.955} C_VEL
LIN {X 0,Y 554.213,Z 365.73,A -85,B 0,C 180,E1 -3168.056,E2 -3168.056} C_VEL
LIN {X 0,Y 551.681,Z 355.236,A -85,B 0,C 180,E1 -3168.339,E2 -3168.339} C_VEL
LIN {X 0,Y 551.719,Z 352.167,A -85,B 0,C 180,E1 -3170.896,E2 -3170.896} C_VEL
LIN {X 0,Y 551.746,Z 349.301,A -85,B 0,C 180,E1 -3173.491,E2 -3173.491} C_VEL
LIN {X 0,Y 551.806,Z 346.243,A -85,B 0,C 180,E1 -3176.472,E2 -3176.472} C_VEL
LIN {X 0,Y 551.805,Z 343.663,A -85,B 0,C 180,E1 -3178.945,E2 -3178.945} C_VEL
LIN {X 0,Y 551.871,Z 341.076,A -85,B 0,C 180,E1 -3181.475,E2 -3181.475} C_VEL
LIN {X 0,Y 551.908,Z 338.442,A -85,B 0,C 180,E1 -3184.136,E2 -3184.136} C_VEL
LIN {X 0,Y 551.935,Z 335.898,A -85,B 0,C 180,E1 -3186.76,E2 -3186.76} C_VEL
LIN {X 0,Y 551.978,Z 333.213,A -85,B 0,C 180,E1 -3189.54,E2 -3189.54} C_VEL
LIN {X 0,Y 551.974,Z 332.358,A -85,B 0,C 180,E1 -3190.493,E2 -3190.493} C_VEL
LIN {X 0,Y 552.128,Z 332.332,A -85,B 0,C 180,E1 -3192.425,E2 -3192.425} C_VEL
LIN {X 0,Y 552.097,Z 332.338,A -85,B 0,C 180,E1 -3195.562,E2 -3195.562} C_VEL
LIN {X 0,Y 552.138,Z 332.333,A -85,B 0,C 180,E1 -3198.676,E2 -3198.676} C_VEL
LIN {X 0,Y 552.12,Z 332.334,A -85,B 0,C 180,E1 -3201.411,E2 -3201.411} C_VEL
LIN {X 0,Y 552.113,Z 332.336,A -85,B 0,C 180,E1 -3204.158,E2 -3204.158} C_VEL
LIN {X 0,Y 552.115,Z 332.337,A -85,B 0,C 180,E1 -3206.814,E2 -3206.814} C_VEL
LIN {X 0,Y 552.113,Z 332.336,A -85,B 0,C 180,E1 -3209.391,E2 -3209.391} C_VEL
LIN {X 0,Y 552.126,Z 332.331,A -85,B 0,C 180,E1 -3211.902,E2 -3211.902} C_VEL
LIN {X 0,Y 552.156,Z 332.331,A -85,B 0,C 180,E1 -3214.649,E2 -3214.649} C_VEL
LIN {X 0,Y 552.095,Z 332.339,A -85,B 0,C 180,E1 -3217.549,E2 -3217.549} C_VEL
LIN {X 0,Y 552.156,Z 332.331,A -85,B 0,C 180,E1 -3220.674,E2 -3220.674} C_VEL
LIN {X 0,Y 552.12,Z 332.336,A -85,B 0,C 180,E1 -3223.737,E2 -3223.737} C_VEL
LIN {X 0,Y 552.136,Z 332.33,A -85,B 0,C 180,E1 -3226.004,E2 -3226.004} C_VEL
LIN {X 0,Y 552.161,Z 332.328,A -85,B 0,C 180,E1 -3228.993,E2 -3228.993} C_VEL
LIN {X 0,Y 552.159,Z 332.329,A -85,B 0,C 180,E1 -3231.951,E2 -3231.951} C_VEL
LIN {X 0,Y 552.229,Z 332.321,A -85,B 0,C 180,E1 -3234.889,E2 -3234.889} C_VEL
LIN {X 0,Y 552.22,Z 332.322,A -85,B 0,C 180,E1 -3237.812,E2 -3237.812} C_VEL
LIN {X 0,Y 552.243,Z 332.32,A -85,B 0,C 180,E1 -3240.729,E2 -3240.729} C_VEL
LIN {X 0,Y 552.208,Z 332.325,A -85,B 0,C 180,E1 -3242.918,E2 -3242.918} C_VEL
LIN {X 0,Y 552.198,Z 332.326,A -85,B 0,C 180,E1 -3245.844,E2 -3245.844} C_VEL
LIN {X 0,Y 552.157,Z 332.33,A -85,B 0,C 180,E1 -3248.786,E2 -3248.786} C_VEL
LIN {X 0,Y 552.163,Z 332.329,A -85,B 0,C 180,E1 -3251.75,E2 -3251.75} C_VEL
LIN {X 0,Y 552.135,Z 332.332,A -85,B 0,C 180,E1 -3254.748,E2 -3254.748} C_VEL
LIN {X 0,Y 552.11,Z 332.335,A -85,B 0,C 180,E1 -3257.788,E2 -3257.788} C_VEL
LIN {X 0,Y 552.129,Z 332.337,A -85,B 0,C 180,E1 -3260.101,E2 -3260.101} C_VEL
LIN {X 0,Y 552.095,Z 332.338,A -85,B 0,C 180,E1 -3262.451,E2 -3262.451} C_VEL
LIN {X 0,Y 552.153,Z 332.331,A -85,B 0,C 180,E1 -3265.35,E2 -3265.35} C_VEL
LIN {X 0,Y 552.121,Z 332.336,A -85,B 0,C 180,E1 -3268.098,E2 -3268.098} C_VEL
LIN {X 0,Y 552.113,Z 332.341,A -85,B 0,C 180,E1 -3270.609,E2 -3270.609} C_VEL
LIN {X 0,Y 552.121,Z 332.335,A -85,B 0,C 180,E1 -3273.185,E2 -3273.185} C_VEL
LIN {X 0,Y 552.112,Z 332.336,A -85,B 0,C 180,E1 -3275.842,E2 -3275.842} C_VEL
LIN {X 0,Y 552.125,Z 332.334,A -85,B 0,C 180,E1 -3279.062,E2 -3279.062} C_VEL
LIN {X 0,Y 552.139,Z 332.337,A -85,B 0,C 180,E1 -3281.444,E2 -3281.444} C_VEL
LIN {X 0,Y 552.093,Z 332.34,A -85,B 0,C 180,E1 -3284.532,E2 -3284.532} C_VEL
LIN {X 0,Y 552.126,Z 332.447,A -85,B 0,C 180,E1 -3286.515,E2 -3286.515} C_VEL
LIN {X 0,Y 552.809,Z 337.039,A -85,B 0,C 180,E1 -3288.618,E2 -3288.618} C_VEL
LIN {X 0,Y 552.76,Z 342.353,A -85,B 0,C 180,E1 -3290.857,E2 -3290.857} C_VEL
LIN {X 0,Y 552.63,Z 349.753,A -85,B 0,C 180,E1 -3293.747,E2 -3293.747} C_VEL
LIN {X 0,Y 552.486,Z 358.08,A -85,B 0,C 180,E1 -3296.84,E2 -3296.84} C_VEL
LIN {X 0,Y 552.403,Z 365.267,A -85,B 0,C 180,E1 -3299.41,E2 -3299.41} C_VEL
LIN {X 0,Y 552.299,Z 373.677,A -85,B 0,C 180,E1 -3302.325,E2 -3302.325} C_VEL
LIN {X 0,Y 552.213,Z 382.121,A -85,B 0,C 180,E1 -3305.166,E2 -3305.166} C_VEL
LIN {X 0,Y 552.118,Z 390.506,A -85,B 0,C 180,E1 -3307.945,E2 -3307.945} C_VEL
LIN {X 0,Y 552.031,Z 398.678,A -85,B 0,C 180,E1 -3310.67,E2 -3310.67} C_VEL
LIN {X 0,Y 552.012,Z 401.748,A -85,B 0,C 180,E1 -3311.68,E2 -3311.68} C_VEL
LIN {X 0,Y 554.455,Z 412.37,A -85,B 0,C 180,E1 -3311.927,E2 -3311.927} C_VEL
LIN {X 0,Y 554.252,Z 428.38,A -85,B 0,C 180,E1 -3312.303,E2 -3312.303} C_VEL
LIN {X 0,Y 554.029,Z 443.653,A -85,B 0,C 180,E1 -3312.825,E2 -3312.825} C_VEL
LIN {X 0,Y 553.675,Z 458.606,A -85,B 0,C 180,E1 -3313.5,E2 -3313.5} C_VEL
LIN {X 0,Y 553.394,Z 471.78,A -85,B 0,C 180,E1 -3314.249,E2 -3314.249} C_VEL
LIN {X 0,Y 553.086,Z 485.301,A -85,B 0,C 180,E1 -3315.193,E2 -3315.193} C_VEL
LIN {X 0,Y 552.716,Z 497.383,A -85,B 0,C 180,E1 -3316.207,E2 -3316.207} C_VEL
LIN {X 0,Y 552.481,Z 508.512,A -85,B 0,C 180,E1 -3317.325,E2 -3317.325} C_VEL
LIN {X 0,Y 552.215,Z 518.487,A -85,B 0,C 180,E1 -3318.514,E2 -3318.514} C_VEL
LIN {X 0,Y 552.124,Z 527.089,A -85,B 0,C 180,E1 -3319.735,E2 -3319.735} C_VEL
LIN {X 0,Y 551.92,Z 534.745,A -85,B 0,C 180,E1 -3321.026,E2 -3321.026} C_VEL
LIN {X 0,Y 551.837,Z 541.091,A -85,B 0,C 180,E1 -3322.315,E2 -3322.315} C_VEL
LIN {X 0,Y 551.769,Z 546.571,A -85,B 0,C 180,E1 -3323.681,E2 -3323.681} C_VEL
LIN {X 0,Y 551.713,Z 550.387,A -85,B 0,C 180,E1 -3324.884,E2 -3324.884} C_VEL
LIN {X 0,Y 551.73,Z 553.89,A -85,B 0,C 180,E1 -3326.349,E2 -3326.349} C_VEL
LIN {X 0,Y 551.655,Z 556.191,A -85,B 0,C 180,E1 -3327.81,E2 -3327.81} C_VEL
LIN {X 0,Y 551.639,Z 557.349,A -85,B 0,C 180,E1 -3329.27,E2 -3329.27} C_VEL
LIN {X 0,Y 551.639,Z 557.348,A -85,B 0,C 180,E1 -3330.73,E2 -3330.73} C_VEL
LIN {X 0,Y 551.655,Z 556.189,A -85,B 0,C 180,E1 -3332.191,E2 -3332.191} C_VEL
LIN {X 0,Y 551.73,Z 553.885,A -85,B 0,C 180,E1 -3333.652,E2 -3333.652} C_VEL
LIN {X 0,Y 551.713,Z 550.385,A -85,B 0,C 180,E1 -3335.116,E2 -3335.116} C_VEL
LIN {X 0,Y 551.821,Z 545.608,A -85,B 0,C 180,E1 -3336.582,E2 -3336.582} C_VEL
LIN {X 0,Y 551.877,Z 539.42,A -85,B 0,C 180,E1 -3338.053,E2 -3338.053} C_VEL
LIN {X 0,Y 551.951,Z 531.644,A -85,B 0,C 180,E1 -3339.528,E2 -3339.528} C_VEL
LIN {X 0,Y 552.185,Z 523.366,A -85,B 0,C 180,E1 -3340.821,E2 -3340.821} C_VEL
LIN {X 0,Y 552.353,Z 513.389,A -85,B 0,C 180,E1 -3342.119,E2 -3342.119} C_VEL
LIN {X 0,Y 552.609,Z 503.184,A -85,B 0,C 180,E1 -3343.234,E2 -3343.234} C_VEL
LIN {X 0,Y 552.889,Z 491.016,A -85,B 0,C 180,E1 -3344.352,E2 -3344.352} C_VEL
LIN {X 0,Y 553.247,Z 478.441,A -85,B 0,C 180,E1 -3345.31,E2 -3345.31} C_VEL
LIN {X 0,Y 553.528,Z 465.505,A -85,B 0,C 180,E1 -3346.126,E2 -3346.126} C_VEL
LIN {X 0,Y 553.856,Z 450.82,A -85,B 0,C 180,E1 -3346.874,E2 -3346.874} C_VEL
LIN {X 0,Y 554.164,Z 435.652,A -85,B 0,C 180,E1 -3347.47,E2 -3347.47} C_VEL
LIN {X 0,Y 554.385,Z 420.423,A -85,B 0,C 180,E1 -3347.904,E2 -3347.904} C_VEL
LIN {X 0,Y 554.348,Z 411.738,A -85,B 0,C 180,E1 -3348.088,E2 -3348.088} C_VEL
LIN {X 0,Y 552.004,Z 401.697,A -85,B 0,C 180,E1 -3348.334,E2 -3348.334} C_VEL
LIN {X 0,Y 552.11,Z 392.838,A -85,B 0,C 180,E1 -3351.272,E2 -3351.272} C_VEL
LIN {X 0,Y 552.175,Z 384.555,A -85,B 0,C 180,E1 -3354.035,E2 -3354.035} C_VEL
LIN {X 0,Y 552.255,Z 377.272,A -85,B 0,C 180,E1 -3356.45,E2 -3356.45} C_VEL
LIN {X 0,Y 552.379,Z 368.85,A -85,B 0,C 180,E1 -3359.33,E2 -3359.33} C_VEL
LIN {X 0,Y 552.47,Z 360.478,A -85,B 0,C 180,E1 -3362.296,E2 -3362.296} C_VEL
LIN {X 0,Y 552.59,Z 351.674,A -85,B 0,C 180,E1 -3365.514,E2 -3365.514} C_VEL
LIN {X 0,Y 552.698,Z 345.301,A -85,B 0,C 180,E1 -3367.966,E2 -3367.966} C_VEL
LIN {X 0,Y 552.835,Z 338.142,A -85,B 0,C 180,E1 -3370.897,E2 -3370.897} C_VEL
LIN {X 0,Y 552.322,Z 333.524,A -85,B 0,C 180,E1 -3372.974,E2 -3372.974} C_VEL
LIN {X 0,Y 552.118,Z 332.337,A -85,B 0,C 180,E1 -3373.582,E2 -3373.582} C_VEL
LIN {X 0,Y 552.108,Z 332.337,A -85,B 0,C 180,E1 -3376.577,E2 -3376.577} C_VEL
LIN {X 0,Y 552.111,Z 332.336,A -85,B 0,C 180,E1 -3379.519,E2 -3379.519} C_VEL
LIN {X 0,Y 552.097,Z 332.339,A -85,B 0,C 180,E1 -3382.337,E2 -3382.337} C_VEL
LIN {X 0,Y 552.132,Z 332.337,A -85,B 0,C 180,E1 -3385.055,E2 -3385.055} C_VEL
LIN {X 0,Y 552.118,Z 332.339,A -85,B 0,C 180,E1 -3387.682,E2 -3387.682} C_VEL
LIN {X 0,Y 552.114,Z 332.335,A -85,B 0,C 180,E1 -3390.235,E2 -3390.235} C_VEL
LIN {X 0,Y 552.142,Z 332.332,A -85,B 0,C 180,E1 -3393,E2 -3393} C_VEL
LIN {X 0,Y 552.116,Z 332.337,A -85,B 0,C 180,E1 -3395.161,E2 -3395.161} C_VEL
LIN {X 0,Y 552.129,Z 332.337,A -85,B 0,C 180,E1 -3398.338,E2 -3398.338} C_VEL
LIN {X 0,Y 552.159,Z 332.329,A -85,B 0,C 180,E1 -3400.675,E2 -3400.675} C_VEL
LIN {X 0,Y 552.12,Z 332.335,A -85,B 0,C 180,E1 -3403.737,E2 -3403.737} C_VEL
LIN {X 0,Y 552.14,Z 332.337,A -85,B 0,C 180,E1 -3406.005,E2 -3406.005} C_VEL
LIN {X 0,Y 552.166,Z 332.333,A -85,B 0,C 180,E1 -3408.994,E2 -3408.994} C_VEL
LIN {X 0,Y 552.162,Z 332.332,A -85,B 0,C 180,E1 -3411.952,E2 -3411.952} C_VEL
LIN {X 0,Y 552.233,Z 332.322,A -85,B 0,C 180,E1 -3414.889,E2 -3414.889} C_VEL
LIN {X 0,Y 552.226,Z 332.322,A -85,B 0,C 180,E1 -3417.812,E2 -3417.812} C_VEL
LIN {X 0,Y 552.247,Z 332.318,A -85,B 0,C 180,E1 -3420.729,E2 -3420.729} C_VEL
LIN {X 0,Y 552.212,Z 332.327,A -85,B 0,C 180,E1 -3422.918,E2 -3422.918} C_VEL
LIN {X 0,Y 552.205,Z 332.329,A -85,B 0,C 180,E1 -3425.844,E2 -3425.844} C_VEL
LIN {X 0,Y 552.166,Z 332.332,A -85,B 0,C 180,E1 -3428.786,E2 -3428.786} C_VEL
LIN {X 0,Y 552.167,Z 332.329,A -85,B 0,C 180,E1 -3431.75,E2 -3431.75} C_VEL
LIN {X 0,Y 552.141,Z 332.331,A -85,B 0,C 180,E1 -3434.748,E2 -3434.748} C_VEL
LIN {X 0,Y 552.117,Z 332.336,A -85,B 0,C 180,E1 -3437.788,E2 -3437.788} C_VEL
LIN {X 0,Y 552.133,Z 332.328,A -85,B 0,C 180,E1 -3440.101,E2 -3440.101} C_VEL
LIN {X 0,Y 552.095,Z 332.338,A -85,B 0,C 180,E1 -3442.451,E2 -3442.451} C_VEL
LIN {X 0,Y 552.16,Z 332.33,A -85,B 0,C 180,E1 -3445.35,E2 -3445.35} C_VEL
LIN {X 0,Y 552.113,Z 332.332,A -85,B 0,C 180,E1 -3448.098,E2 -3448.098} C_VEL
LIN {X 0,Y 552.108,Z 332.338,A -85,B 0,C 180,E1 -3450.61,E2 -3450.61} C_VEL
LIN {X 0,Y 552.119,Z 332.336,A -85,B 0,C 180,E1 -3453.186,E2 -3453.186} C_VEL
LIN {X 0,Y 552.114,Z 332.332,A -85,B 0,C 180,E1 -3453.789,E2 -3453.789} C_VEL
LIN {X 0,Y 551.482,Z 332.413,A -85,B 0,C 180,E1 -3454.397,E2 -3454.397} C_VEL
LIN {X 0,Y 548.665,Z 332.765,A -85,B 0,C 180,E1 -3455.386,E2 -3455.386} C_VEL
LIN {X 0,Y 546.245,Z 333.069,A -85,B 0,C 180,E1 -3456.181,E2 -3456.181} C_VEL
LIN {X 0,Y 545.175,Z 333.201,A -85,B 0,C 180,E1 -3456.795,E2 -3456.795} C_VEL
LIN {X 0,Y 545.072,Z 333.212,A -85,B 0,C 180,E1 -3457.003,E2 -3457.003} C_VEL
LIN {X 0,Y 545.075,Z 333.212,A -85,B 0,C 180,E1 -3460.142,E2 -3460.142} C_VEL
LIN {X 0,Y 545.081,Z 333.212,A -85,B 0,C 180,E1 -3463.106,E2 -3463.106} C_VEL
LIN {X 0,Y 545.07,Z 333.214,A -85,B 0,C 180,E1 -3466.224,E2 -3466.224} C_VEL
LIN {X 0,Y 544.988,Z 333.229,A -85,B 0,C 180,E1 -3468.876,E2 -3468.876} C_VEL
LIN {X 0,Y 544.893,Z 333.253,A -85,B 0,C 180,E1 -3469.842,E2 -3469.842} C_VEL
LIN {X 0,Y 544.878,Z 335.956,A -85,B 0,C 180,E1 -3472.683,E2 -3472.683} C_VEL
LIN {X 0,Y 544.851,Z 338.808,A -85,B 0,C 180,E1 -3475.643,E2 -3475.643} C_VEL
LIN {X 0,Y 544.795,Z 341.477,A -85,B 0,C 180,E1 -3478.366,E2 -3478.366} C_VEL
LIN {X 0,Y 544.766,Z 343.774,A -85,B 0,C 180,E1 -3480.644,E2 -3480.644} C_VEL
LIN {X 0,Y 544.755,Z 346.329,A -85,B 0,C 180,E1 -3483.157,E2 -3483.157} C_VEL
LIN {X 0,Y 544.669,Z 348.902,A -85,B 0,C 180,E1 -3485.612,E2 -3485.612} C_VEL
LIN {X 0,Y 544.642,Z 352.25,A -85,B 0,C 180,E1 -3488.819,E2 -3488.819} C_VEL
LIN {X 0,Y 544.606,Z 355.294,A -85,B 0,C 180,E1 -3491.517,E2 -3491.517} C_VEL
LIN {X 0,Y 547.615,Z 368.348,A -85,B 0,C 180,E1 -3491.865,E2 -3491.865} C_VEL
LIN {X 0,Y 547.395,Z 383.58,A -85,B 0,C 180,E1 -3492.284,E2 -3492.284} C_VEL
LIN {X 0,Y 547.104,Z 397.622,A -85,B 0,C 180,E1 -3492.815,E2 -3492.815} C_VEL
LIN {X 0,Y 546.787,Z 411.288,A -85,B 0,C 180,E1 -3493.478,E2 -3493.478} C_VEL
LIN {X 0,Y 546.393,Z 425.374,A -85,B 0,C 180,E1 -3494.329,E2 -3494.329} C_VEL
LIN {X 0,Y 546.046,Z 438.147,A -85,B 0,C 180,E1 -3495.274,E2 -3495.274} C_VEL
LIN {X 0,Y 545.727,Z 448.866,A -85,B 0,C 180,E1 -3496.217,E2 -3496.217} C_VEL
LIN {X 0,Y 545.453,Z 459.748,A -85,B 0,C 180,E1 -3497.347,E2 -3497.347} C_VEL
LIN {X 0,Y 545.171,Z 469.886,A -85,B 0,C 180,E1 -3498.599,E2 -3498.599} C_VEL
LIN {X 0,Y 544.987,Z 479.143,A -85,B 0,C 180,E1 -3499.974,E2 -3499.974} C_VEL
LIN {X 0,Y 544.847,Z 485.501,A -85,B 0,C 180,E1 -3501.095,E2 -3501.095} C_VEL
LIN {X 0,Y 544.747,Z 492.505,A -85,B 0,C 180,E1 -3502.587,E2 -3502.587} C_VEL
LIN {X 0,Y 544.703,Z 498.014,A -85,B 0,C 180,E1 -3504.075,E2 -3504.075} C_VEL
LIN {X 0,Y 544.606,Z 502.18,A -85,B 0,C 180,E1 -3505.559,E2 -3505.559} C_VEL
LIN {X 0,Y 544.643,Z 505.113,A -85,B 0,C 180,E1 -3507.041,E2 -3507.041} C_VEL
LIN {X 0,Y 544.543,Z 506.879,A -85,B 0,C 180,E1 -3508.521,E2 -3508.521} C_VEL
LIN {X 0,Y 544.539,Z 507.496,A -85,B 0,C 180,E1 -3510,E2 -3510} C_VEL
LIN {X 0,Y 544.545,Z 506.939,A -85,B 0,C 180,E1 -3511.479,E2 -3511.479} C_VEL
LIN {X 0,Y 544.645,Z 505.254,A -85,B 0,C 180,E1 -3512.958,E2 -3512.958} C_VEL
LIN {X 0,Y 544.605,Z 502.401,A -85,B 0,C 180,E1 -3514.44,E2 -3514.44} C_VEL
LIN {X 0,Y 544.696,Z 498.313,A -85,B 0,C 180,E1 -3515.924,E2 -3515.924} C_VEL
LIN {X 0,Y 544.746,Z 492.897,A -85,B 0,C 180,E1 -3517.412,E2 -3517.412} C_VEL
LIN {X 0,Y 544.845,Z 485.994,A -85,B 0,C 180,E1 -3518.904,E2 -3518.904} C_VEL
LIN {X 0,Y 545.081,Z 477.383,A -85,B 0,C 180,E1 -3520.399,E2 -3520.399} C_VEL
LIN {X 0,Y 545.231,Z 467.754,A -85,B 0,C 180,E1 -3521.774,E2 -3521.774} C_VEL
LIN {X 0,Y 545.53,Z 457.175,A -85,B 0,C 180,E1 -3523.029,E2 -3523.029} C_VEL
LIN {X 0,Y 545.829,Z 445.799,A -85,B 0,C 180,E1 -3524.16,E2 -3524.16} C_VEL
LIN {X 0,Y 546.15,Z 433.586,A -85,B 0,C 180,E1 -3525.177,E2 -3525.177} C_VEL
LIN {X 0,Y 546.521,Z 420.992,A -85,B 0,C 180,E1 -3526.05,E2 -3526.05} C_VEL
LIN {X 0,Y 546.873,Z 407.663,A -85,B 0,C 180,E1 -3526.807,E2 -3526.807} C_VEL
LIN {X 0,Y 547.227,Z 394.24,A -85,B 0,C 180,E1 -3527.415,E2 -3527.415} C_VEL
LIN {X 0,Y 547.454,Z 379.844,A -85,B 0,C 180,E1 -3527.922,E2 -3527.922} C_VEL
LIN {X 0,Y 547.591,Z 367.619,A -85,B 0,C 180,E1 -3528.241,E2 -3528.241} C_VEL
LIN {X 0,Y 544.591,Z 355.234,A -85,B 0,C 180,E1 -3528.587,E2 -3528.587} C_VEL
LIN {X 0,Y 544.649,Z 351.765,A -85,B 0,C 180,E1 -3531.71,E2 -3531.71} C_VEL
LIN {X 0,Y 544.666,Z 348.964,A -85,B 0,C 180,E1 -3534.387,E2 -3534.387} C_VEL
LIN {X 0,Y 544.726,Z 346.197,A -85,B 0,C 180,E1 -3537.098,E2 -3537.098} C_VEL
LIN {X 0,Y 544.796,Z 343.003,A -85,B 0,C 180,E1 -3540.206,E2 -3540.206} C_VEL
LIN {X 0,Y 544.827,Z 340.192,A -85,B 0,C 180,E1 -3543.021,E2 -3543.021} C_VEL
LIN {X 0,Y 544.87,Z 337.659,A -85,B 0,C 180,E1 -3545.649,E2 -3545.649} C_VEL
LIN {X 0,Y 544.9,Z 335.163,A -85,B 0,C 180,E1 -3548.249,E2 -3548.249} C_VEL
LIN {X 0,Y 544.926,Z 333.235,A -85,B 0,C 180,E1 -3550.453,E2 -3550.453} C_VEL
LIN {X 0,Y 545.086,Z 333.215,A -85,B 0,C 180,E1 -3553.105,E2 -3553.105} C_VEL
LIN {X 0,Y 545.066,Z 333.217,A -85,B 0,C 180,E1 -3556.224,E2 -3556.224} C_VEL
LIN {X 0,Y 545.095,Z 333.212,A -85,B 0,C 180,E1 -3558.886,E2 -3558.886} C_VEL
LIN {X 0,Y 545.054,Z 333.215,A -85,B 0,C 180,E1 -3561.763,E2 -3561.763} C_VEL
LIN {X 0,Y 545.065,Z 333.213,A -85,B 0,C 180,E1 -3564.534,E2 -3564.534} C_VEL
LIN {X 0,Y 545.068,Z 333.211,A -85,B 0,C 180,E1 -3567.211,E2 -3567.211} C_VEL
LIN {X 0,Y 545.101,Z 333.214,A -85,B 0,C 180,E1 -3569.813,E2 -3569.813} C_VEL
LIN {X 0,Y 545.101,Z 333.209,A -85,B 0,C 180,E1 -3572.824,E2 -3572.824} C_VEL
LIN {X 0,Y 545.052,Z 333.217,A -85,B 0,C 180,E1 -3575.631,E2 -3575.631} C_VEL
LIN {X 0,Y 545.065,Z 333.214,A -85,B 0,C 180,E1 -3578.837,E2 -3578.837} C_VEL
LIN {X 0,Y 545.082,Z 333.209,A -85,B 0,C 180,E1 -3581.196,E2 -3581.196} C_VEL
LIN {X 0,Y 545.076,Z 333.216,A -85,B 0,C 180,E1 -3583.521,E2 -3583.521} C_VEL
LIN {X 0,Y 545.095,Z 333.206,A -85,B 0,C 180,E1 -3585.82,E2 -3585.82} C_VEL
LIN {X 0,Y 545.116,Z 333.205,A -85,B 0,C 180,E1 -3588.849,E2 -3588.849} C_VEL
LIN {X 0,Y 545.129,Z 333.205,A -85,B 0,C 180,E1 -3591.847,E2 -3591.847} C_VEL
LIN {X 0,Y 545.205,Z 333.196,A -85,B 0,C 180,E1 -3594.823,E2 -3594.823} C_VEL
LIN {X 0,Y 545.193,Z 333.197,A -85,B 0,C 180,E1 -3597.784,E2 -3597.784} C_VEL
LIN {X 0,Y 545.213,Z 333.195,A -85,B 0,C 180,E1 -3600.739,E2 -3600.739} C_VEL
LIN {X 0,Y 545.174,Z 333.201,A -85,B 0,C 180,E1 -3602.956,E2 -3602.956} C_VEL
LIN {X 0,Y 545.17,Z 333.202,A -85,B 0,C 180,E1 -3605.919,E2 -3605.919} C_VEL
LIN {X 0,Y 545.117,Z 333.208,A -85,B 0,C 180,E1 -3608.9,E2 -3608.9} C_VEL
LIN {X 0,Y 545.135,Z 333.205,A -85,B 0,C 180,E1 -3611.904,E2 -3611.904} C_VEL
LIN {X 0,Y 545.084,Z 333.211,A -85,B 0,C 180,E1 -3614.944,E2 -3614.944} C_VEL
LIN {X 0,Y 545.078,Z 333.212,A -85,B 0,C 180,E1 -3618.026,E2 -3618.026} C_VEL
LIN {X 0,Y 545.093,Z 333.211,A -85,B 0,C 180,E1 -3620.372,E2 -3620.372} C_VEL
LIN {X 0,Y 545.09,Z 333.211,A -85,B 0,C 180,E1 -3623.559,E2 -3623.559} C_VEL
LIN {X 0,Y 545.078,Z 333.216,A -85,B 0,C 180,E1 -3626.001,E2 -3626.001} C_VEL
LIN {X 0,Y 545.09,Z 333.212,A -85,B 0,C 180,E1 -3628.749,E2 -3628.749} C_VEL
LIN {X 0,Y 545.076,Z 333.213,A -85,B 0,C 180,E1 -3631.683,E2 -3631.683} C_VEL
LIN {X 0,Y 545.08,Z 333.212,A -85,B 0,C 180,E1 -3634.563,E2 -3634.563} C_VEL
LIN {X 0,Y 545.038,Z 333.218,A -85,B 0,C 180,E1 -3637.304,E2 -3637.304} C_VEL
LIN {X 0,Y 545.074,Z 333.215,A -85,B 0,C 180,E1 -3640.142,E2 -3640.142} C_VEL
LIN {X 0,Y 545.061,Z 333.216,A -85,B 0,C 180,E1 -3642.697,E2 -3642.697} C_VEL
LIN {X 0,Y 545.077,Z 333.217,A -85,B 0,C 180,E1 -3645.873,E2 -3645.873} C_VEL
LIN {X 0,Y 545.121,Z 333.276,A -85,B 0,C 180,E1 -3646.218,E2 -3646.218} C_VEL
LIN {X 0,Y 545.779,Z 337.785,A -85,B 0,C 180,E1 -3648.319,E2 -3648.319} C_VEL
LIN {X 0,Y 545.82,Z 341.466,A -85,B 0,C 180,E1 -3649.925,E2 -3649.925} C_VEL
LIN {X 0,Y 545.662,Z 348.438,A -85,B 0,C 180,E1 -3652.747,E2 -3652.747} C_VEL
LIN {X 0,Y 545.516,Z 355.731,A -85,B 0,C 180,E1 -3655.54,E2 -3655.54} C_VEL
LIN {X 0,Y 545.418,Z 363.119,A -85,B 0,C 180,E1 -3658.26,E2 -3658.26} C_VEL
LIN {X 0,Y 545.302,Z 371.399,A -85,B 0,C 180,E1 -3661.211,E2 -3661.211} C_VEL
LIN {X 0,Y 545.196,Z 379.463,A -85,B 0,C 180,E1 -3664.006,E2 -3664.006} C_VEL
LIN {X 0,Y 545.081,Z 387.959,A -85,B 0,C 180,E1 -3666.843,E2 -3666.843} C_VEL
LIN {X 0,Y 545.023,Z 396.343,A -85,B 0,C 180,E1 -3669.625,E2 -3669.625} C_VEL
LIN {X 0,Y 544.946,Z 401.722,A -85,B 0,C 180,E1 -3671.428,E2 -3671.428} C_VEL
LIN {X 0,Y 547.698,Z 413.712,A -85,B 0,C 180,E1 -3671.724,E2 -3671.724} C_VEL
LIN {X 0,Y 547.485,Z 428.889,A -85,B 0,C 180,E1 -3672.093,E2 -3672.093} C_VEL
LIN {X 0,Y 547.277,Z 442.92,A -85,B 0,C 180,E1 -3672.575,E2 -3672.575} C_VEL
LIN {X 0,Y 546.903,Z 456.785,A -85,B 0,C 180,E1 -3673.194,E2 -3673.194} C_VEL
LIN {X 0,Y 546.574,Z 470.256,A -85,B 0,C 180,E1 -3673.952,E2 -3673.952} C_VEL
LIN {X 0,Y 546.228,Z 482.537,A -85,B 0,C 180,E1 -3674.792,E2 -3674.792} C_VEL
LIN {X 0,Y 545.847,Z 495.297,A -85,B 0,C 180,E1 -3675.84,E2 -3675.84} C_VEL
LIN {X 0,Y 545.567,Z 506.753,A -85,B 0,C 180,E1 -3676.972,E2 -3676.972} C_VEL
LIN {X 0,Y 545.281,Z 516.392,A -85,B 0,C 180,E1 -3678.099,E2 -3678.099} C_VEL
LIN {X 0,Y 545.086,Z 525.857,A -85,B 0,C 180,E1 -3679.413,E2 -3679.413} C_VEL
LIN {X 0,Y 544.899,Z 533.737,A -85,B 0,C 180,E1 -3680.722,E2 -3680.722} C_VEL
LIN {X 0,Y 544.771,Z 541.091,A -85,B 0,C 180,E1 -3682.215,E2 -3682.215} C_VEL
LIN {X 0,Y 544.675,Z 546.917,A -85,B 0,C 180,E1 -3683.702,E2 -3683.702} C_VEL
LIN {X 0,Y 544.642,Z 550.387,A -85,B 0,C 180,E1 -3684.818,E2 -3684.818} C_VEL
LIN {X 0,Y 544.644,Z 553.889,A -85,B 0,C 180,E1 -3686.301,E2 -3686.301} C_VEL
LIN {X 0,Y 544.569,Z 556.191,A -85,B 0,C 180,E1 -3687.781,E2 -3687.781} C_VEL
LIN {X 0,Y 544.539,Z 557.348,A -85,B 0,C 180,E1 -3689.261,E2 -3689.261} C_VEL
LIN {X 0,Y 544.539,Z 557.348,A -85,B 0,C 180,E1 -3690.74,E2 -3690.74} C_VEL
LIN {X 0,Y 544.569,Z 556.188,A -85,B 0,C 180,E1 -3692.219,E2 -3692.219} C_VEL
LIN {X 0,Y 544.644,Z 553.885,A -85,B 0,C 180,E1 -3693.7,E2 -3693.7} C_VEL
LIN {X 0,Y 544.642,Z 550.386,A -85,B 0,C 180,E1 -3695.183,E2 -3695.183} C_VEL
LIN {X 0,Y 544.753,Z 545.608,A -85,B 0,C 180,E1 -3696.668,E2 -3696.668} C_VEL
LIN {X 0,Y 544.819,Z 539.42,A -85,B 0,C 180,E1 -3698.158,E2 -3698.158} C_VEL
LIN {X 0,Y 544.904,Z 531.643,A -85,B 0,C 180,E1 -3699.653,E2 -3699.653} C_VEL
LIN {X 0,Y 545.151,Z 523.365,A -85,B 0,C 180,E1 -3700.962,E2 -3700.962} C_VEL
LIN {X 0,Y 545.358,Z 513.389,A -85,B 0,C 180,E1 -3702.277,E2 -3702.277} C_VEL
LIN {X 0,Y 545.639,Z 503.183,A -85,B 0,C 180,E1 -3703.406,E2 -3703.406} C_VEL
LIN {X 0,Y 545.971,Z 491.015,A -85,B 0,C 180,E1 -3704.538,E2 -3704.538} C_VEL
LIN {X 0,Y 546.354,Z 478.64,A -85,B 0,C 180,E1 -3705.493,E2 -3705.493} C_VEL
LIN {X 0,Y 546.667,Z 465.503,A -85,B 0,C 180,E1 -3706.334,E2 -3706.334} C_VEL
LIN {X 0,Y 547.046,Z 450.818,A -85,B 0,C 180,E1 -3707.091,E2 -3707.091} C_VEL
LIN {X 0,Y 547.371,Z 436.398,A -85,B 0,C 180,E1 -3707.666,E2 -3707.666} C_VEL
LIN {X 0,Y 547.592,Z 421.892,A -85,B 0,C 180,E1 -3708.095,E2 -3708.095} C_VEL
LIN {X 0,Y 547.572,Z 412.779,A -85,B 0,C 180,E1 -3708.3,E2 -3708.3} C_VEL
LIN {X 0,Y 544.946,Z 401.732,A -85,B 0,C 180,E1 -3708.569,E2 -3708.569} C_VEL
LIN {X 0,Y 545.069,Z 393.017,A -85,B 0,C 180,E1 -3711.492,E2 -3711.492} C_VEL
LIN {X 0,Y 545.131,Z 384.314,A -85,B 0,C 180,E1 -3714.366,E2 -3714.366} C_VEL
LIN {X 0,Y 545.274,Z 375.915,A -85,B 0,C 180,E1 -3717.21,E2 -3717.21} C_VEL
LIN {X 0,Y 545.321,Z 367.458,A -85,B 0,C 180,E1 -3720.174,E2 -3720.174} C_VEL
LIN {X 0,Y 545.454,Z 360.305,A -85,B 0,C 180,E1 -3722.763,E2 -3722.763} C_VEL
LIN {X 0,Y 545.607,Z 352.266,A -85,B 0,C 180,E1 -3725.757,E2 -3725.757} C_VEL
LIN {X 0,Y 545.74,Z 344.91,A -85,B 0,C 180,E1 -3728.651,E2 -3728.651} C_VEL
LIN {X 0,Y 545.857,Z 339.194,A -85,B 0,C 180,E1 -3731.044,E2 -3731.044} C_VEL
LIN {X 0,Y 545.332,Z 334.741,A -85,B 0,C 180,E1 -3733.082,E2 -3733.082} C_VEL
LIN {X 0,Y 545.108,Z 333.208,A -85,B 0,C 180,E1 -3733.921,E2 -3733.921} C_VEL
LIN {X 0,Y 545.08,Z 333.215,A -85,B 0,C 180,E1 -3736.894,E2 -3736.894} C_VEL
LIN {X 0,Y 545.069,Z 333.215,A -85,B 0,C 180,E1 -3739.858,E2 -3739.858} C_VEL
LIN {X 0,Y 545.078,Z 333.217,A -85,B 0,C 180,E1 -3743.073,E2 -3743.073} C_VEL
LIN {X 0,Y 545.088,Z 333.212,A -85,B 0,C 180,E1 -3745.606,E2 -3745.606} C_VEL
LIN {X 0,Y 545.06,Z 333.215,A -85,B 0,C 180,E1 -3748.321,E2 -3748.321} C_VEL
LIN {X 0,Y 545.092,Z 333.211,A -85,B 0,C 180,E1 -3751.252,E2 -3751.252} C_VEL
LIN {X 0,Y 545.081,Z 333.216,A -85,B 0,C 180,E1 -3754,E2 -3754} C_VEL
LIN {X 0,Y 545.082,Z 333.212,A -85,B 0,C 180,E1 -3756.441,E2 -3756.441} C_VEL
LIN {X 0,Y 545.098,Z 333.211,A -85,B 0,C 180,E1 -3759.628,E2 -3759.628} C_VEL
LIN {X 0,Y 545.098,Z 333.211,A -85,B 0,C 180,E1 -3762.75,E2 -3762.75} C_VEL
LIN {X 0,Y 545.099,Z 333.212,A -85,B 0,C 180,E1 -3765.82,E2 -3765.82} C_VEL
LIN {X 0,Y 545.122,Z 333.209,A -85,B 0,C 180,E1 -3768.85,E2 -3768.85} C_VEL
LIN {X 0,Y 545.132,Z 333.207,A -85,B 0,C 180,E1 -3771.847,E2 -3771.847} C_VEL
LIN {X 0,Y 545.208,Z 333.196,A -85,B 0,C 180,E1 -3774.823,E2 -3774.823} C_VEL
LIN {X 0,Y 545.198,Z 333.197,A -85,B 0,C 180,E1 -3777.784,E2 -3777.784} C_VEL
LIN {X 0,Y 545.217,Z 333.194,A -85,B 0,C 180,E1 -3780.739,E2 -3780.739} C_VEL
LIN {X 0,Y 545.178,Z 333.203,A -85,B 0,C 180,E1 -3782.956,E2 -3782.956} C_VEL
LIN {X 0,Y 545.177,Z 333.204,A -85,B 0,C 180,E1 -3785.92,E2 -3785.92} C_VEL
LIN {X 0,Y 545.125,Z 333.211,A -85,B 0,C 180,E1 -3788.9,E2 -3788.9} C_VEL
LIN {X 0,Y 545.139,Z 333.205,A -85,B 0,C 180,E1 -3791.904,E2 -3791.904} C_VEL
LIN {X 0,Y 545.09,Z 333.212,A -85,B 0,C 180,E1 -3794.944,E2 -3794.944} C_VEL
LIN {X 0,Y 545.084,Z 333.215,A -85,B 0,C 180,E1 -3798.026,E2 -3798.026} C_VEL
LIN {X 0,Y 545.098,Z 333.202,A -85,B 0,C 180,E1 -3800.372,E2 -3800.372} C_VEL
LIN {X 0,Y 545.083,Z 333.211,A -85,B 0,C 180,E1 -3803.559,E2 -3803.559} C_VEL
LIN {X 0,Y 545.084,Z 333.21,A -85,B 0,C 180,E1 -3806,E2 -3806} C_VEL
LIN {X 0,Y 545.093,Z 333.212,A -85,B 0,C 180,E1 -3808.748,E2 -3808.748} C_VEL
LIN {X 0,Y 545.061,Z 333.217,A -85,B 0,C 180,E1 -3811.679,E2 -3811.679} C_VEL
LIN {X 0,Y 545.081,Z 333.211,A -85,B 0,C 180,E1 -3814.563,E2 -3814.563} C_VEL
LIN {X 0,Y 545.072,Z 333.212,A -85,B 0,C 180,E1 -3817.003,E2 -3817.003} C_VEL
LIN {X 0,Y 544.362,Z 333.305,A -85,B 0,C 180,E1 -3817.619,E2 -3817.619} C_VEL
LIN {X 0,Y 541.496,Z 333.658,A -85,B 0,C 180,E1 -3818.62,E2 -3818.62} C_VEL
LIN {X 0,Y 539.109,Z 333.96,A -85,B 0,C 180,E1 -3819.426,E2 -3819.426} C_VEL
LIN {X 0,Y 538.099,Z 334.082,A -85,B 0,C 180,E1 -3820.048,E2 -3820.048} C_VEL
LIN {X 0,Y 538.024,Z 334.091,A -85,B 0,C 180,E1 -3820.258,E2 -3820.258} C_VEL
LIN {X 0,Y 538.029,Z 334.091,A -85,B 0,C 180,E1 -3822.987,E2 -3822.987} C_VEL
LIN {X 0,Y 538.033,Z 334.092,A -85,B 0,C 180,E1 -3825.925,E2 -3825.925} C_VEL
LIN {X 0,Y 538.003,Z 334.096,A -85,B 0,C 180,E1 -3828.224,E2 -3828.224} C_VEL
LIN {X 0,Y 537.836,Z 334.314,A -85,B 0,C 180,E1 -3830.186,E2 -3830.186} C_VEL
LIN {X 0,Y 537.823,Z 337.012,A -85,B 0,C 180,E1 -3833.051,E2 -3833.051} C_VEL
LIN {X 0,Y 537.772,Z 339.649,A -85,B 0,C 180,E1 -3835.809,E2 -3835.809} C_VEL
LIN {X 0,Y 537.74,Z 342.237,A -85,B 0,C 180,E1 -3838.481,E2 -3838.481} C_VEL
LIN {X 0,Y 537.686,Z 344.899,A -85,B 0,C 180,E1 -3841.134,E2 -3841.134} C_VEL
LIN {X 0,Y 537.654,Z 347.419,A -85,B 0,C 180,E1 -3843.613,E2 -3843.613} C_VEL
LIN {X 0,Y 537.621,Z 350.118,A -85,B 0,C 180,E1 -3846.216,E2 -3846.216} C_VEL
LIN {X 0,Y 537.576,Z 352.545,A -85,B 0,C 180,E1 -3848.527,E2 -3848.527} C_VEL
LIN {X 0,Y 537.521,Z 355.433,A -85,B 0,C 180,E1 -3851.264,E2 -3851.264} C_VEL
LIN {X 0,Y 540.857,Z 369.043,A -85,B 0,C 180,E1 -3851.644,E2 -3851.644} C_VEL
LIN {X 0,Y 540.614,Z 384.538,A -85,B 0,C 180,E1 -3852.084,E2 -3852.084} C_VEL
LIN {X 0,Y 540.267,Z 399.877,A -85,B 0,C 180,E1 -3852.688,E2 -3852.688} C_VEL
LIN {X 0,Y 539.866,Z 414.767,A -85,B 0,C 180,E1 -3853.455,E2 -3853.455} C_VEL
LIN {X 0,Y 539.469,Z 428.196,A -85,B 0,C 180,E1 -3854.316,E2 -3854.316} C_VEL
LIN {X 0,Y 539.027,Z 441.588,A -85,B 0,C 180,E1 -3855.367,E2 -3855.367} C_VEL
LIN {X 0,Y 538.666,Z 452.757,A -85,B 0,C 180,E1 -3856.417,E2 -3856.417} C_VEL
LIN {X 0,Y 538.367,Z 463.007,A -85,B 0,C 180,E1 -3857.561,E2 -3857.561} C_VEL
LIN {X 0,Y 538.122,Z 473.047,A -85,B 0,C 180,E1 -3858.893,E2 -3858.893} C_VEL
LIN {X 0,Y 537.874,Z 481.378,A -85,B 0,C 180,E1 -3860.22,E2 -3860.22} C_VEL
LIN {X 0,Y 537.737,Z 489.204,A -85,B 0,C 180,E1 -3861.734,E2 -3861.734} C_VEL
LIN {X 0,Y 537.621,Z 495.438,A -85,B 0,C 180,E1 -3863.243,E2 -3863.243} C_VEL
LIN {X 0,Y 537.574,Z 500.259,A -85,B 0,C 180,E1 -3864.749,E2 -3864.749} C_VEL
LIN {X 0,Y 537.562,Z 503.796,A -85,B 0,C 180,E1 -3866.252,E2 -3866.252} C_VEL
LIN {X 0,Y 537.488,Z 506.139,A -85,B 0,C 180,E1 -3867.752,E2 -3867.752} C_VEL
LIN {X 0,Y 537.437,Z 507.337,A -85,B 0,C 180,E1 -3869.25,E2 -3869.25} C_VEL
LIN {X 0,Y 537.439,Z 507.358,A -85,B 0,C 180,E1 -3870.749,E2 -3870.749} C_VEL
LIN {X 0,Y 537.488,Z 506.238,A -85,B 0,C 180,E1 -3872.248,E2 -3872.248} C_VEL
LIN {X 0,Y 537.562,Z 503.975,A -85,B 0,C 180,E1 -3873.748,E2 -3873.748} C_VEL
LIN {X 0,Y 537.572,Z 500.515,A -85,B 0,C 180,E1 -3875.25,E2 -3875.25} C_VEL
LIN {X 0,Y 537.619,Z 495.777,A -85,B 0,C 180,E1 -3876.756,E2 -3876.756} C_VEL
LIN {X 0,Y 537.735,Z 489.64,A -85,B 0,C 180,E1 -3878.265,E2 -3878.265} C_VEL
LIN {X 0,Y 537.858,Z 481.915,A -85,B 0,C 180,E1 -3879.78,E2 -3879.78} C_VEL
LIN {X 0,Y 538.081,Z 473.677,A -85,B 0,C 180,E1 -3881.107,E2 -3881.107} C_VEL
LIN {X 0,Y 538.347,Z 463.764,A -85,B 0,C 180,E1 -3882.439,E2 -3882.439} C_VEL
LIN {X 0,Y 538.645,Z 453.604,A -85,B 0,C 180,E1 -3883.583,E2 -3883.583} C_VEL
LIN {X 0,Y 538.997,Z 441.515,A -85,B 0,C 180,E1 -3884.729,E2 -3884.729} C_VEL
LIN {X 0,Y 539.446,Z 429.313,A -85,B 0,C 180,E1 -3885.691,E2 -3885.691} C_VEL
LIN {X 0,Y 539.815,Z 416.248,A -85,B 0,C 180,E1 -3886.546,E2 -3886.546} C_VEL
LIN {X 0,Y 540.147,Z 403.734,A -85,B 0,C 180,E1 -3887.218,E2 -3887.218} C_VEL
LIN {X 0,Y 540.543,Z 388.796,A -85,B 0,C 180,E1 -3887.851,E2 -3887.851} C_VEL
LIN {X 0,Y 540.796,Z 374.415,A -85,B 0,C 180,E1 -3888.308,E2 -3888.308} C_VEL
LIN {X 0,Y 540.839,Z 368.927,A -85,B 0,C 180,E1 -3888.448,E2 -3888.448} C_VEL
LIN {X 0,Y 537.543,Z 355.383,A -85,B 0,C 180,E1 -3888.847,E2 -3888.847} C_VEL
LIN {X 0,Y 537.592,Z 352.223,A -85,B 0,C 180,E1 -3891.845,E2 -3891.845} C_VEL
LIN {X 0,Y 537.616,Z 349.212,A -85,B 0,C 180,E1 -3894.728,E2 -3894.728} C_VEL
LIN {X 0,Y 537.654,Z 346.613,A -85,B 0,C 180,E1 -3897.268,E2 -3897.268} C_VEL
LIN {X 0,Y 537.715,Z 343.45,A -85,B 0,C 180,E1 -3900.387,E2 -3900.387} C_VEL
LIN {X 0,Y 537.774,Z 340.598,A -85,B 0,C 180,E1 -3903.29,E2 -3903.29} C_VEL
LIN {X 0,Y 537.801,Z 337.989,A -85,B 0,C 180,E1 -3906.019,E2 -3906.019} C_VEL
LIN {X 0,Y 537.823,Z 335.322,A -85,B 0,C 180,E1 -3908.846,E2 -3908.846} C_VEL
LIN {X 0,Y 537.843,Z 334.404,A -85,B 0,C 180,E1 -3909.812,E2 -3909.812} C_VEL
LIN {X 0,Y 537.999,Z 334.094,A -85,B 0,C 180,E1 -3911.875,E2 -3911.875} C_VEL
LIN {X 0,Y 538.032,Z 334.091,A -85,B 0,C 180,E1 -3914.859,E2 -3914.859} C_VEL
LIN {X 0,Y 538.036,Z 334.089,A -85,B 0,C 180,E1 -3918.12,E2 -3918.12} C_VEL
LIN {X 0,Y 538.039,Z 334.091,A -85,B 0,C 180,E1 -3920.414,E2 -3920.414} C_VEL
LIN {X 0,Y 538.032,Z 334.089,A -85,B 0,C 180,E1 -3923.068,E2 -3923.068} C_VEL
LIN {X 0,Y 538.026,Z 334.088,A -85,B 0,C 180,E1 -3925.827,E2 -3925.827} C_VEL
LIN {X 0,Y 538.022,Z 334.093,A -85,B 0,C 180,E1 -3928.499,E2 -3928.499} C_VEL
LIN {X 0,Y 538.058,Z 334.089,A -85,B 0,C 180,E1 -3931.1,E2 -3931.1} C_VEL
LIN {X 0,Y 538.049,Z 334.083,A -85,B 0,C 180,E1 -3933.634,E2 -3933.634} C_VEL
LIN {X 0,Y 538.022,Z 334.093,A -85,B 0,C 180,E1 -3936.118,E2 -3936.118} C_VEL
LIN {X 0,Y 538.038,Z 334.083,A -85,B 0,C 180,E1 -3939.349,E2 -3939.349} C_VEL
LIN {X 0,Y 538.072,Z 334.084,A -85,B 0,C 180,E1 -3942.517,E2 -3942.517} C_VEL
LIN {X 0,Y 538.063,Z 334.082,A -85,B 0,C 180,E1 -3945.631,E2 -3945.631} C_VEL
LIN {X 0,Y 538.076,Z 334.082,A -85,B 0,C 180,E1 -3948.701,E2 -3948.701} C_VEL
LIN {X 0,Y 538.086,Z 334.082,A -85,B 0,C 180,E1 -3951.74,E2 -3951.74} C_VEL
LIN {X 0,Y 538.163,Z 334.073,A -85,B 0,C 180,E1 -3954.755,E2 -3954.755} C_VEL
LIN {X 0,Y 538.165,Z 334.073,A -85,B 0,C 180,E1 -3957.755,E2 -3957.755} C_VEL
LIN {X 0,Y 538.183,Z 334.071,A -85,B 0,C 180,E1 -3960.748,E2 -3960.748} C_VEL
LIN {X 0,Y 538.141,Z 334.078,A -85,B 0,C 180,E1 -3962.994,E2 -3962.994} C_VEL
LIN {X 0,Y 538.123,Z 334.08,A -85,B 0,C 180,E1 -3965.997,E2 -3965.997} C_VEL
LIN {X 0,Y 538.068,Z 334.086,A -85,B 0,C 180,E1 -3969.018,E2 -3969.018} C_VEL
LIN {X 0,Y 538.083,Z 334.084,A -85,B 0,C 180,E1 -3972.062,E2 -3972.062} C_VEL
LIN {X 0,Y 538.044,Z 334.089,A -85,B 0,C 180,E1 -3975.144,E2 -3975.144} C_VEL
LIN {X 0,Y 538.03,Z 334.092,A -85,B 0,C 180,E1 -3978.27,E2 -3978.27} C_VEL
LIN {X 0,Y 538.038,Z 334.088,A -85,B 0,C 180,E1 -3980.651,E2 -3980.651} C_VEL
LIN {X 0,Y 538.022,Z 334.091,A -85,B 0,C 180,E1 -3983.887,E2 -3983.887} C_VEL
LIN {X 0,Y 538.041,Z 334.092,A -85,B 0,C 180,E1 -3986.367,E2 -3986.367} C_VEL
LIN {X 0,Y 538.035,Z 334.093,A -85,B 0,C 180,E1 -3988.935,E2 -3988.935} C_VEL
LIN {X 0,Y 538.026,Z 334.093,A -85,B 0,C 180,E1 -3991.89,E2 -3991.89} C_VEL
LIN {X 0,Y 538.03,Z 334.091,A -85,B 0,C 180,E1 -3994.621,E2 -3994.621} C_VEL
LIN {X 0,Y 538.007,Z 334.094,A -85,B 0,C 180,E1 -3997.171,E2 -3997.171} C_VEL
LIN {X 0,Y 538.029,Z 334.095,A -85,B 0,C 180,E1 -3999.796,E2 -3999.796} C_VEL
LIN {X 0,Y 538.017,Z 334.093,A -85,B 0,C 180,E1 -4002.786,E2 -4002.786} C_VEL
LIN {X 0,Y 538.055,Z 334.135,A -85,B 0,C 180,E1 -4005.923,E2 -4005.923} C_VEL
LIN {X 0,Y 538.825,Z 339.147,A -85,B 0,C 180,E1 -4008.303,E2 -4008.303} C_VEL
LIN {X 0,Y 538.869,Z 342.52,A -85,B 0,C 180,E1 -4009.791,E2 -4009.791} C_VEL
LIN {X 0,Y 538.672,Z 349.702,A -85,B 0,C 180,E1 -4012.736,E2 -4012.736} C_VEL
LIN {X 0,Y 538.529,Z 356.29,A -85,B 0,C 180,E1 -4015.303,E2 -4015.303} C_VEL
LIN {X 0,Y 538.443,Z 363.596,A -85,B 0,C 180,E1 -4018.039,E2 -4018.039} C_VEL
LIN {X 0,Y 538.285,Z 372.099,A -85,B 0,C 180,E1 -4021.114,E2 -4021.114} C_VEL
LIN {X 0,Y 538.187,Z 379.254,A -85,B 0,C 180,E1 -4023.641,E2 -4023.641} C_VEL
LIN {X 0,Y 538.05,Z 387.71,A -85,B 0,C 180,E1 -4026.523,E2 -4026.523} C_VEL
LIN {X 0,Y 537.97,Z 396.173,A -85,B 0,C 180,E1 -4029.346,E2 -4029.346} C_VEL
LIN {X 0,Y 537.892,Z 401.73,A -85,B 0,C 180,E1 -4031.178,E2 -4031.178} C_VEL
LIN {X 0,Y 540.939,Z 415.171,A -85,B 0,C 180,E1 -4031.519,E2 -4031.519} C_VEL
LIN {X 0,Y 540.689,Z 430.452,A -85,B 0,C 180,E1 -4031.911,E2 -4031.911} C_VEL
LIN {X 0,Y 540.441,Z 445.035,A -85,B 0,C 180,E1 -4032.439,E2 -4032.439} C_VEL
LIN {X 0,Y 540.035,Z 458.602,A -85,B 0,C 180,E1 -4033.071,E2 -4033.071} C_VEL
LIN {X 0,Y 539.663,Z 471.775,A -85,B 0,C 180,E1 -4033.838,E2 -4033.838} C_VEL
LIN {X 0,Y 539.259,Z 485.544,A -85,B 0,C 180,E1 -4034.825,E2 -4034.825} C_VEL
LIN {X 0,Y 538.851,Z 497.38,A -85,B 0,C 180,E1 -4035.845,E2 -4035.845} C_VEL
LIN {X 0,Y 538.525,Z 508.511,A -85,B 0,C 180,E1 -4036.99,E2 -4036.99} C_VEL
LIN {X 0,Y 538.178,Z 518.732,A -85,B 0,C 180,E1 -4038.242,E2 -4038.242} C_VEL
LIN {X 0,Y 538.017,Z 528.298,A -85,B 0,C 180,E1 -4039.653,E2 -4039.653} C_VEL
LIN {X 0,Y 537.797,Z 535.752,A -85,B 0,C 180,E1 -4040.978,E2 -4040.978} C_VEL
LIN {X 0,Y 537.661,Z 542.702,A -85,B 0,C 180,E1 -4042.489,E2 -4042.489} C_VEL
LIN {X 0,Y 537.623,Z 548.164,A -85,B 0,C 180,E1 -4043.997,E2 -4043.997} C_VEL
LIN {X 0,Y 537.507,Z 552.292,A -85,B 0,C 180,E1 -4045.501,E2 -4045.501} C_VEL
LIN {X 0,Y 537.544,Z 555.186,A -85,B 0,C 180,E1 -4047.003,E2 -4047.003} C_VEL
LIN {X 0,Y 537.449,Z 556.91,A -85,B 0,C 180,E1 -4048.502,E2 -4048.502} C_VEL
LIN {X 0,Y 537.439,Z 557.5,A -85,B 0,C 180,E1 -4050,E2 -4050} C_VEL
LIN {X 0,Y 537.449,Z 556.908,A -85,B 0,C 180,E1 -4051.499,E2 -4051.499} C_VEL
LIN {X 0,Y 537.544,Z 555.181,A -85,B 0,C 180,E1 -4052.998,E2 -4052.998} C_VEL
LIN {X 0,Y 537.507,Z 552.288,A -85,B 0,C 180,E1 -4054.5,E2 -4054.5} C_VEL
LIN {X 0,Y 537.623,Z 548.164,A -85,B 0,C 180,E1 -4056.003,E2 -4056.003} C_VEL
LIN {X 0,Y 537.661,Z 542.7,A -85,B 0,C 180,E1 -4057.511,E2 -4057.511} C_VEL
LIN {X 0,Y 537.797,Z 535.743,A -85,B 0,C 180,E1 -4059.023,E2 -4059.023} C_VEL
LIN {X 0,Y 538.024,Z 527.081,A -85,B 0,C 180,E1 -4060.538,E2 -4060.538} C_VEL
LIN {X 0,Y 538.229,Z 517.531,A -85,B 0,C 180,E1 -4061.912,E2 -4061.912} C_VEL
LIN {X 0,Y 538.525,Z 508.505,A -85,B 0,C 180,E1 -4063.01,E2 -4063.01} C_VEL
LIN {X 0,Y 538.838,Z 496.355,A -85,B 0,C 180,E1 -4064.252,E2 -4064.252} C_VEL
LIN {X 0,Y 539.284,Z 484.496,A -85,B 0,C 180,E1 -4065.261,E2 -4065.261} C_VEL
LIN {X 0,Y 539.664,Z 471.764,A -85,B 0,C 180,E1 -4066.163,E2 -4066.163} C_VEL
LIN {X 0,Y 540.044,Z 458.583,A -85,B 0,C 180,E1 -4066.929,E2 -4066.929} C_VEL
LIN {X 0,Y 540.409,Z 445.027,A -85,B 0,C 180,E1 -4067.563,E2 -4067.563} C_VEL
LIN {X 0,Y 540.689,Z 430.469,A -85,B 0,C 180,E1 -4068.089,E2 -4068.089} C_VEL
LIN {X 0,Y 540.954,Z 414.931,A -85,B 0,C 180,E1 -4068.486,E2 -4068.486} C_VEL
LIN {X 0,Y 537.887,Z 401.729,A -85,B 0,C 180,E1 -4068.822,E2 -4068.822} C_VEL
LIN {X 0,Y 537.999,Z 393.733,A -85,B 0,C 180,E1 -4071.455,E2 -4071.455} C_VEL
LIN {X 0,Y 538.09,Z 384.071,A -85,B 0,C 180,E1 -4074.706,E2 -4074.706} C_VEL
LIN {X 0,Y 538.238,Z 376.299,A -85,B 0,C 180,E1 -4077.389,E2 -4077.389} C_VEL
LIN {X 0,Y 538.3,Z 368.627,A -85,B 0,C 180,E1 -4080.122,E2 -4080.122} C_VEL
LIN {X 0,Y 538.448,Z 361.328,A -85,B 0,C 180,E1 -4082.798,E2 -4082.798} C_VEL
LIN {X 0,Y 538.617,Z 354.171,A -85,B 0,C 180,E1 -4085.496,E2 -4085.496} C_VEL
LIN {X 0,Y 538.759,Z 346.628,A -85,B 0,C 180,E1 -4088.493,E2 -4088.493} C_VEL
LIN {X 0,Y 538.867,Z 341.032,A -85,B 0,C 180,E1 -4090.848,E2 -4090.848} C_VEL
LIN {X 0,Y 538.51,Z 336.902,A -85,B 0,C 180,E1 -4092.738,E2 -4092.738} C_VEL
LIN {X 0,Y 538.044,Z 334.087,A -85,B 0,C 180,E1 -4094.183,E2 -4094.183} C_VEL
LIN {X 0,Y 538.021,Z 334.095,A -85,B 0,C 180,E1 -4097.214,E2 -4097.214} C_VEL
LIN {X 0,Y 538.027,Z 334.095,A -85,B 0,C 180,E1 -4100.203,E2 -4100.203} C_VEL
LIN {X 0,Y 538.032,Z 334.095,A -85,B 0,C 180,E1 -4103.068,E2 -4103.068} C_VEL
LIN {X 0,Y 538.029,Z 334.092,A -85,B 0,C 180,E1 -4105.828,E2 -4105.828} C_VEL
LIN {X 0,Y 538.011,Z 334.092,A -85,B 0,C 180,E1 -4108.499,E2 -4108.499} C_VEL
LIN {X 0,Y 538.063,Z 334.089,A -85,B 0,C 180,E1 -4111.1,E2 -4111.1} C_VEL
LIN {X 0,Y 538.044,Z 334.09,A -85,B 0,C 180,E1 -4113.634,E2 -4113.634} C_VEL
LIN {X 0,Y 538.01,Z 334.092,A -85,B 0,C 180,E1 -4116.122,E2 -4116.122} C_VEL
LIN {X 0,Y 538.042,Z 334.088,A -85,B 0,C 180,E1 -4119.349,E2 -4119.349} C_VEL
LIN {X 0,Y 538.058,Z 334.087,A -85,B 0,C 180,E1 -4122.517,E2 -4122.517} C_VEL
LIN {X 0,Y 538.068,Z 334.086,A -85,B 0,C 180,E1 -4125.631,E2 -4125.631} C_VEL
LIN {X 0,Y 538.081,Z 334.085,A -85,B 0,C 180,E1 -4128.702,E2 -4128.702} C_VEL
LIN {X 0,Y 538.089,Z 334.083,A -85,B 0,C 180,E1 -4131.74,E2 -4131.74} C_VEL
LIN {X 0,Y 538.165,Z 334.073,A -85,B 0,C 180,E1 -4134.755,E2 -4134.755} C_VEL
LIN {X 0,Y 538.17,Z 334.072,A -85,B 0,C 180,E1 -4137.755,E2 -4137.755} C_VEL
LIN {X 0,Y 538.187,Z 334.07,A -85,B 0,C 180,E1 -4140.748,E2 -4140.748} C_VEL
LIN {X 0,Y 538.144,Z 334.078,A -85,B 0,C 180,E1 -4142.995,E2 -4142.995} C_VEL
LIN {X 0,Y 538.13,Z 334.08,A -85,B 0,C 180,E1 -4145.997,E2 -4145.997} C_VEL
LIN {X 0,Y 538.075,Z 334.088,A -85,B 0,C 180,E1 -4149.018,E2 -4149.018} C_VEL
LIN {X 0,Y 538.087,Z 334.08,A -85,B 0,C 180,E1 -4152.063,E2 -4152.063} C_VEL
LIN {X 0,Y 538.049,Z 334.091,A -85,B 0,C 180,E1 -4155.144,E2 -4155.144} C_VEL
LIN {X 0,Y 538.036,Z 334.09,A -85,B 0,C 180,E1 -4158.27,E2 -4158.27} C_VEL
LIN {X 0,Y 538.043,Z 334.081,A -85,B 0,C 180,E1 -4160.651,E2 -4160.651} C_VEL
LIN {X 0,Y 538.006,Z 334.094,A -85,B 0,C 180,E1 -4163.888,E2 -4163.888} C_VEL
LIN {X 0,Y 538.046,Z 334.084,A -85,B 0,C 180,E1 -4166.367,E2 -4166.367} C_VEL
LIN {X 0,Y 538.034,Z 334.092,A -85,B 0,C 180,E1 -4168.933,E2 -4168.933} C_VEL
LIN {X 0,Y 538.014,Z 334.094,A -85,B 0,C 180,E1 -4171.887,E2 -4171.887} C_VEL
LIN {X 0,Y 538.03,Z 334.089,A -85,B 0,C 180,E1 -4174.62,E2 -4174.62} C_VEL
LIN {X 0,Y 538.013,Z 334.092,A -85,B 0,C 180,E1 -4177.171,E2 -4177.171} C_VEL
LIN {X 0,Y 538.024,Z 334.091,A -85,B 0,C 180,E1 -4180.258,E2 -4180.258} C_VEL
LIN {X 0,Y 537.374,Z 334.176,A -85,B 0,C 180,E1 -4180.884,E2 -4180.884} C_VEL
LIN {X 0,Y 534.524,Z 334.531,A -85,B 0,C 180,E1 -4181.898,E2 -4181.898} C_VEL
LIN {X 0,Y 532.101,Z 334.832,A -85,B 0,C 180,E1 -4182.716,E2 -4182.716} C_VEL
LIN {X 0,Y 531.053,Z 334.961,A -85,B 0,C 180,E1 -4183.347,E2 -4183.347} C_VEL
LIN {X 0,Y 530.965,Z 334.97,A -85,B 0,C 180,E1 -4183.56,E2 -4183.56} C_VEL
LIN {X 0,Y 530.968,Z 334.971,A -85,B 0,C 180,E1 -4186.505,E2 -4186.505} C_VEL
LIN {X 0,Y 530.868,Z 334.988,A -85,B 0,C 180,E1 -4188.991,E2 -4188.991} C_VEL
LIN {X 0,Y 530.79,Z 335.034,A -85,B 0,C 180,E1 -4190.171,E2 -4190.171} C_VEL
LIN {X 0,Y 530.749,Z 337.307,A -85,B 0,C 180,E1 -4192.608,E2 -4192.608} C_VEL
LIN {X 0,Y 530.751,Z 339.839,A -85,B 0,C 180,E1 -4195.292,E2 -4195.292} C_VEL
LIN {X 0,Y 530.677,Z 342.441,A -85,B 0,C 180,E1 -4198.012,E2 -4198.012} C_VEL
LIN {X 0,Y 530.629,Z 345.32,A -85,B 0,C 180,E1 -4200.944,E2 -4200.944} C_VEL
LIN {X 0,Y 530.587,Z 348.677,A -85,B 0,C 180,E1 -4204.252,E2 -4204.252} C_VEL
LIN {X 0,Y 530.505,Z 351.081,A -85,B 0,C 180,E1 -4206.582,E2 -4206.582} C_VEL
LIN {X 0,Y 530.491,Z 353.69,A -85,B 0,C 180,E1 -4209.041,E2 -4209.041} C_VEL
LIN {X 0,Y 530.463,Z 355.719,A -85,B 0,C 180,E1 -4211.003,E2 -4211.003} C_VEL
LIN {X 0,Y 534.154,Z 370.27,A -85,B 0,C 180,E1 -4211.427,E2 -4211.427} C_VEL
LIN {X 0,Y 533.866,Z 384.929,A -85,B 0,C 180,E1 -4211.854,E2 -4211.854} C_VEL
LIN {X 0,Y 533.482,Z 400.067,A -85,B 0,C 180,E1 -4212.461,E2 -4212.461} C_VEL
LIN {X 0,Y 533.056,Z 414.871,A -85,B 0,C 180,E1 -4213.237,E2 -4213.237} C_VEL
LIN {X 0,Y 532.578,Z 428.416,A -85,B 0,C 180,E1 -4214.123,E2 -4214.123} C_VEL
LIN {X 0,Y 532.079,Z 441.593,A -85,B 0,C 180,E1 -4215.172,E2 -4215.172} C_VEL
LIN {X 0,Y 531.716,Z 452.762,A -85,B 0,C 180,E1 -4216.236,E2 -4216.236} C_VEL
LIN {X 0,Y 531.389,Z 463.012,A -85,B 0,C 180,E1 -4217.395,E2 -4217.395} C_VEL
LIN {X 0,Y 531.091,Z 473.05,A -85,B 0,C 180,E1 -4218.744,E2 -4218.744} C_VEL
LIN {X 0,Y 530.821,Z 481.38,A -85,B 0,C 180,E1 -4220.089,E2 -4220.089} C_VEL
LIN {X 0,Y 530.668,Z 489.206,A -85,B 0,C 180,E1 -4221.623,E2 -4221.623} C_VEL
LIN {X 0,Y 530.552,Z 495.44,A -85,B 0,C 180,E1 -4223.153,E2 -4223.153} C_VEL
LIN {X 0,Y 530.508,Z 500.26,A -85,B 0,C 180,E1 -4224.679,E2 -4224.679} C_VEL
LIN {X 0,Y 530.481,Z 503.797,A -85,B 0,C 180,E1 -4226.202,E2 -4226.202} C_VEL
LIN {X 0,Y 530.409,Z 506.138,A -85,B 0,C 180,E1 -4227.722,E2 -4227.722} C_VEL
LIN {X 0,Y 530.34,Z 507.337,A -85,B 0,C 180,E1 -4229.24,E2 -4229.24} C_VEL
LIN {X 0,Y 530.341,Z 507.357,A -85,B 0,C 180,E1 -4230.759,E2 -4230.759} C_VEL
LIN {X 0,Y 530.41,Z 506.237,A -85,B 0,C 180,E1 -4232.278,E2 -4232.278} C_VEL
LIN {X 0,Y 530.481,Z 503.974,A -85,B 0,C 180,E1 -4233.798,E2 -4233.798} C_VEL
LIN {X 0,Y 530.506,Z 500.513,A -85,B 0,C 180,E1 -4235.321,E2 -4235.321} C_VEL
LIN {X 0,Y 530.55,Z 495.774,A -85,B 0,C 180,E1 -4236.847,E2 -4236.847} C_VEL
LIN {X 0,Y 530.665,Z 489.637,A -85,B 0,C 180,E1 -4238.376,E2 -4238.376} C_VEL
LIN {X 0,Y 530.808,Z 481.911,A -85,B 0,C 180,E1 -4239.911,E2 -4239.911} C_VEL
LIN {X 0,Y 531.04,Z 473.673,A -85,B 0,C 180,E1 -4241.257,E2 -4241.257} C_VEL
LIN {X 0,Y 531.347,Z 463.759,A -85,B 0,C 180,E1 -4242.605,E2 -4242.605} C_VEL
LIN {X 0,Y 531.702,Z 453.597,A -85,B 0,C 180,E1 -4243.764,E2 -4243.764} C_VEL
LIN {X 0,Y 532.088,Z 441.506,A -85,B 0,C 180,E1 -4244.925,E2 -4244.925} C_VEL
LIN {X 0,Y 532.612,Z 428.235,A -85,B 0,C 180,E1 -4245.979,E2 -4245.979} C_VEL
LIN {X 0,Y 533.048,Z 414.752,A -85,B 0,C 180,E1 -4246.861,E2 -4246.861} C_VEL
LIN {X 0,Y 533.465,Z 400.91,A -85,B 0,C 180,E1 -4247.588,E2 -4247.588} C_VEL
LIN {X 0,Y 533.818,Z 385.777,A -85,B 0,C 180,E1 -4248.207,E2 -4248.207} C_VEL
LIN {X 0,Y 534.115,Z 370.16,A -85,B 0,C 180,E1 -4248.667,E2 -4248.667} C_VEL
LIN {X 0,Y 530.459,Z 355.725,A -85,B 0,C 180,E1 -4249.092,E2 -4249.092} C_VEL
LIN {X 0,Y 530.509,Z 352.692,A -85,B 0,C 180,E1 -4251.976,E2 -4251.976} C_VEL
LIN {X 0,Y 530.517,Z 350.313,A -85,B 0,C 180,E1 -4254.247,E2 -4254.247} C_VEL
LIN {X 0,Y 530.568,Z 347.732,A -85,B 0,C 180,E1 -4256.767,E2 -4256.767} C_VEL
LIN {X 0,Y 530.604,Z 345.122,A -85,B 0,C 180,E1 -4259.345,E2 -4259.345} C_VEL
LIN {X 0,Y 530.671,Z 342.477,A -85,B 0,C 180,E1 -4262.049,E2 -4262.049} C_VEL
LIN {X 0,Y 530.726,Z 339.83,A -85,B 0,C 180,E1 -4264.813,E2 -4264.813} C_VEL
LIN {X 0,Y 530.748,Z 337.271,A -85,B 0,C 180,E1 -4267.525,E2 -4267.525} C_VEL
LIN {X 0,Y 530.797,Z 335.12,A -85,B 0,C 180,E1 -4269.83,E2 -4269.83} C_VEL
LIN {X 0,Y 530.971,Z 334.968,A -85,B 0,C 180,E1 -4272.457,E2 -4272.457} C_VEL
LIN {X 0,Y 530.987,Z 334.967,A -85,B 0,C 180,E1 -4275.62,E2 -4275.62} C_VEL
LIN {X 0,Y 530.999,Z 334.966,A -85,B 0,C 180,E1 -4278.565,E2 -4278.565} C_VEL
LIN {X 0,Y 530.959,Z 334.97,A -85,B 0,C 180,E1 -4281.529,E2 -4281.529} C_VEL
LIN {X 0,Y 530.982,Z 334.967,A -85,B 0,C 180,E1 -4284.382,E2 -4284.382} C_VEL
LIN {X 0,Y 530.967,Z 334.967,A -85,B 0,C 180,E1 -4287.133,E2 -4287.133} C_VEL
LIN {X 0,Y 530.986,Z 334.972,A -85,B 0,C 180,E1 -4289.804,E2 -4289.804} C_VEL
LIN {X 0,Y 531.017,Z 334.961,A -85,B 0,C 180,E1 -4292.466,E2 -4292.466} C_VEL
LIN {X 0,Y 531.007,Z 334.964,A -85,B 0,C 180,E1 -4294.942,E2 -4294.942} C_VEL
LIN {X 0,Y 530.97,Z 334.966,A -85,B 0,C 180,E1 -4298.247,E2 -4298.247} C_VEL
LIN {X 0,Y 530.996,Z 334.966,A -85,B 0,C 180,E1 -4300.677,E2 -4300.677} C_VEL
LIN {X 0,Y 530.992,Z 334.967,A -85,B 0,C 180,E1 -4303.071,E2 -4303.071} C_VEL
LIN {X 0,Y 531.018,Z 334.96,A -85,B 0,C 180,E1 -4305.436,E2 -4305.436} C_VEL
LIN {X 0,Y 531.047,Z 334.958,A -85,B 0,C 180,E1 -4308.55,E2 -4308.55} C_VEL
LIN {X 0,Y 531.056,Z 334.958,A -85,B 0,C 180,E1 -4311.629,E2 -4311.629} C_VEL
LIN {X 0,Y 531.122,Z 334.951,A -85,B 0,C 180,E1 -4314.685,E2 -4314.685} C_VEL
LIN {X 0,Y 531.137,Z 334.949,A -85,B 0,C 180,E1 -4317.725,E2 -4317.725} C_VEL
LIN {X 0,Y 531.153,Z 334.947,A -85,B 0,C 180,E1 -4320.758,E2 -4320.758} C_VEL
LIN {X 0,Y 531.107,Z 334.954,A -85,B 0,C 180,E1 -4323.034,E2 -4323.034} C_VEL
LIN {X 0,Y 531.082,Z 334.958,A -85,B 0,C 180,E1 -4326.077,E2 -4326.077} C_VEL
LIN {X 0,Y 531.028,Z 334.965,A -85,B 0,C 180,E1 -4329.138,E2 -4329.138} C_VEL
LIN {X 0,Y 531.04,Z 334.963,A -85,B 0,C 180,E1 -4332.225,E2 -4332.225} C_VEL
LIN {X 0,Y 530.994,Z 334.97,A -85,B 0,C 180,E1 -4335.35,E2 -4335.35} C_VEL
LIN {X 0,Y 530.989,Z 334.971,A -85,B 0,C 180,E1 -4338.521,E2 -4338.521} C_VEL
LIN {X 0,Y 530.998,Z 334.965,A -85,B 0,C 180,E1 -4340.938,E2 -4340.938} C_VEL
LIN {X 0,Y 530.978,Z 334.97,A -85,B 0,C 180,E1 -4344.224,E2 -4344.224} C_VEL
LIN {X 0,Y 531.004,Z 334.966,A -85,B 0,C 180,E1 -4346.744,E2 -4346.744} C_VEL
LIN {X 0,Y 530.991,Z 334.97,A -85,B 0,C 180,E1 -4349.322,E2 -4349.322} C_VEL
LIN {X 0,Y 530.978,Z 334.972,A -85,B 0,C 180,E1 -4352.103,E2 -4352.103} C_VEL
LIN {X 0,Y 530.987,Z 334.969,A -85,B 0,C 180,E1 -4354.854,E2 -4354.854} C_VEL
LIN {X 0,Y 530.965,Z 334.97,A -85,B 0,C 180,E1 -4357.508,E2 -4357.508} C_VEL
LIN {X 0,Y 530.983,Z 334.969,A -85,B 0,C 180,E1 -4360.433,E2 -4360.433} C_VEL
LIN {X 0,Y 530.965,Z 334.973,A -85,B 0,C 180,E1 -4363.282,E2 -4363.282} C_VEL
LIN {X 0,Y 530.999,Z 334.994,A -85,B 0,C 180,E1 -4365.62,E2 -4365.62} C_VEL
LIN {X 0,Y 531.689,Z 339.362,A -85,B 0,C 180,E1 -4367.75,E2 -4367.75} C_VEL
LIN {X 0,Y 531.932,Z 343.582,A -85,B 0,C 180,E1 -4369.655,E2 -4369.655} C_VEL
LIN {X 0,Y 531.69,Z 350.535,A -85,B 0,C 180,E1 -4372.553,E2 -4372.553} C_VEL
LIN {X 0,Y 531.56,Z 356.835,A -85,B 0,C 180,E1 -4375.058,E2 -4375.058} C_VEL
LIN {X 0,Y 531.414,Z 364.751,A -85,B 0,C 180,E1 -4378.062,E2 -4378.062} C_VEL
LIN {X 0,Y 531.273,Z 372.263,A -85,B 0,C 180,E1 -4380.819,E2 -4380.819} C_VEL
LIN {X 0,Y 531.147,Z 380.249,A -85,B 0,C 180,E1 -4383.688,E2 -4383.688} C_VEL
LIN {X 0,Y 530.968,Z 388.638,A -85,B 0,C 180,E1 -4386.604,E2 -4386.604} C_VEL
LIN {X 0,Y 530.882,Z 397.096,A -85,B 0,C 180,E1 -4389.463,E2 -4389.463} C_VEL
LIN {X 0,Y 530.827,Z 401.497,A -85,B 0,C 180,E1 -4390.919,E2 -4390.919} C_VEL
LIN {X 0,Y 534.197,Z 416.393,A -85,B 0,C 180,E1 -4391.306,E2 -4391.306} C_VEL
LIN {X 0,Y 533.937,Z 431.381,A -85,B 0,C 180,E1 -4391.706,E2 -4391.706} C_VEL
LIN {X 0,Y 533.668,Z 445.181,A -85,B 0,C 180,E1 -4392.215,E2 -4392.215} C_VEL
LIN {X 0,Y 533.223,Z 458.6,A -85,B 0,C 180,E1 -4392.848,E2 -4392.848} C_VEL
LIN {X 0,Y 532.826,Z 471.773,A -85,B 0,C 180,E1 -4393.625,E2 -4393.625} C_VEL
LIN {X 0,Y 532.361,Z 485.228,A -85,B 0,C 180,E1 -4394.597,E2 -4394.597} C_VEL
LIN {X 0,Y 531.921,Z 497.378,A -85,B 0,C 180,E1 -4395.657,E2 -4395.657} C_VEL
LIN {X 0,Y 531.563,Z 508.511,A -85,B 0,C 180,E1 -4396.817,E2 -4396.817} C_VEL
LIN {X 0,Y 531.152,Z 519.273,A -85,B 0,C 180,E1 -4398.16,E2 -4398.16} C_VEL
LIN {X 0,Y 530.979,Z 528.298,A -85,B 0,C 180,E1 -4399.514,E2 -4399.514} C_VEL
LIN {X 0,Y 530.759,Z 535.751,A -85,B 0,C 180,E1 -4400.857,E2 -4400.857} C_VEL
LIN {X 0,Y 530.6,Z 542.702,A -85,B 0,C 180,E1 -4402.389,E2 -4402.389} C_VEL
LIN {X 0,Y 530.528,Z 548.164,A -85,B 0,C 180,E1 -4403.917,E2 -4403.917} C_VEL
LIN {X 0,Y 530.412,Z 552.292,A -85,B 0,C 180,E1 -4405.44,E2 -4405.44} C_VEL
LIN {X 0,Y 530.449,Z 555.185,A -85,B 0,C 180,E1 -4406.962,E2 -4406.962} C_VEL
LIN {X 0,Y 530.359,Z 556.91,A -85,B 0,C 180,E1 -4408.482,E2 -4408.482} C_VEL
LIN {X 0,Y 530.34,Z 557.5,A -85,B 0,C 180,E1 -4410,E2 -4410} C_VEL
LIN {X 0,Y 530.359,Z 556.907,A -85,B 0,C 180,E1 -4411.519,E2 -4411.519} C_VEL
LIN {X 0,Y 530.449,Z 555.18,A -85,B 0,C 180,E1 -4413.038,E2 -4413.038} C_VEL
LIN {X 0,Y 530.412,Z 552.288,A -85,B 0,C 180,E1 -4414.56,E2 -4414.56} C_VEL
LIN {X 0,Y 530.533,Z 548.164,A -85,B 0,C 180,E1 -4416.084,E2 -4416.084} C_VEL
LIN {X 0,Y 530.601,Z 542.699,A -85,B 0,C 180,E1 -4417.612,E2 -4417.612} C_VEL
LIN {X 0,Y 530.76,Z 535.742,A -85,B 0,C 180,E1 -4419.143,E2 -4419.143} C_VEL
LIN {X 0,Y 530.98,Z 528.291,A -85,B 0,C 180,E1 -4420.486,E2 -4420.486} C_VEL
LIN {X 0,Y 531.173,Z 518.955,A -85,B 0,C 180,E1 -4421.884,E2 -4421.884} C_VEL
LIN {X 0,Y 531.564,Z 508.505,A -85,B 0,C 180,E1 -4423.184,E2 -4423.184} C_VEL
LIN {X 0,Y 531.921,Z 496.357,A -85,B 0,C 180,E1 -4424.441,E2 -4424.441} C_VEL
LIN {X 0,Y 532.388,Z 484.121,A -85,B 0,C 180,E1 -4425.493,E2 -4425.493} C_VEL
LIN {X 0,Y 532.823,Z 471.761,A -85,B 0,C 180,E1 -4426.376,E2 -4426.376} C_VEL
LIN {X 0,Y 533.229,Z 458.58,A -85,B 0,C 180,E1 -4427.152,E2 -4427.152} C_VEL
LIN {X 0,Y 533.633,Z 445.181,A -85,B 0,C 180,E1 -4427.786,E2 -4427.786} C_VEL
LIN {X 0,Y 533.934,Z 430.366,A -85,B 0,C 180,E1 -4428.328,E2 -4428.328} C_VEL
LIN {X 0,Y 534.105,Z 415.305,A -85,B 0,C 180,E1 -4428.721,E2 -4428.721} C_VEL
LIN {X 0,Y 530.833,Z 401.459,A -85,B 0,C 180,E1 -4429.093,E2 -4429.093} C_VEL
LIN {X 0,Y 530.937,Z 392.447,A -85,B 0,C 180,E1 -4432.091,E2 -4432.091} C_VEL
LIN {X 0,Y 531.072,Z 383.827,A -85,B 0,C 180,E1 -4435.055,E2 -4435.055} C_VEL
LIN {X 0,Y 531.208,Z 375.451,A -85,B 0,C 180,E1 -4438.013,E2 -4438.013} C_VEL
LIN {X 0,Y 531.332,Z 368.048,A -85,B 0,C 180,E1 -4440.71,E2 -4440.71} C_VEL
LIN {X 0,Y 531.457,Z 362.345,A -85,B 0,C 180,E1 -4442.833,E2 -4442.833} C_VEL
LIN {X 0,Y 531.62,Z 355.204,A -85,B 0,C 180,E1 -4445.569,E2 -4445.569} C_VEL
LIN {X 0,Y 531.783,Z 347.296,A -85,B 0,C 180,E1 -4448.763,E2 -4448.763} C_VEL
LIN {X 0,Y 531.88,Z 341.283,A -85,B 0,C 180,E1 -4451.352,E2 -4451.352} C_VEL
LIN {X 0,Y 531.21,Z 335.997,A -85,B 0,C 180,E1 -4453.859,E2 -4453.859} C_VEL
LIN {X 0,Y 531.001,Z 334.965,A -85,B 0,C 180,E1 -4454.381,E2 -4454.381} C_VEL
LIN {X 0,Y 530.98,Z 334.971,A -85,B 0,C 180,E1 -4457.544,E2 -4457.544} C_VEL
LIN {X 0,Y 530.99,Z 334.97,A -85,B 0,C 180,E1 -4460.557,E2 -4460.557} C_VEL
LIN {X 0,Y 530.976,Z 334.971,A -85,B 0,C 180,E1 -4463.843,E2 -4463.843} C_VEL
LIN {X 0,Y 531.002,Z 334.969,A -85,B 0,C 180,E1 -4466.494,E2 -4466.494} C_VEL
LIN {X 0,Y 530.977,Z 334.972,A -85,B 0,C 180,E1 -4469.355,E2 -4469.355} C_VEL
LIN {X 0,Y 531.018,Z 334.968,A -85,B 0,C 180,E1 -4472.467,E2 -4472.467} C_VEL
LIN {X 0,Y 531.008,Z 334.965,A -85,B 0,C 180,E1 -4474.943,E2 -4474.943} C_VEL
LIN {X 0,Y 530.974,Z 334.971,A -85,B 0,C 180,E1 -4478.247,E2 -4478.247} C_VEL
LIN {X 0,Y 530.998,Z 334.965,A -85,B 0,C 180,E1 -4480.677,E2 -4480.677} C_VEL
LIN {X 0,Y 530.99,Z 334.972,A -85,B 0,C 180,E1 -4483.071,E2 -4483.071} C_VEL
LIN {X 0,Y 531.023,Z 334.963,A -85,B 0,C 180,E1 -4485.436,E2 -4485.436} C_VEL
LIN {X 0,Y 531.041,Z 334.961,A -85,B 0,C 180,E1 -4488.55,E2 -4488.55} C_VEL
LIN {X 0,Y 531.059,Z 334.959,A -85,B 0,C 180,E1 -4491.63,E2 -4491.63} C_VEL
LIN {X 0,Y 531.124,Z 334.95,A -85,B 0,C 180,E1 -4494.685,E2 -4494.685} C_VEL
LIN {X 0,Y 531.142,Z 334.948,A -85,B 0,C 180,E1 -4497.725,E2 -4497.725} C_VEL
LIN {X 0,Y 531.157,Z 334.945,A -85,B 0,C 180,E1 -4500.758,E2 -4500.758} C_VEL
LIN {X 0,Y 531.11,Z 334.954,A -85,B 0,C 180,E1 -4503.034,E2 -4503.034} C_VEL
LIN {X 0,Y 531.09,Z 334.956,A -85,B 0,C 180,E1 -4506.077,E2 -4506.077} C_VEL
LIN {X 0,Y 531.035,Z 334.964,A -85,B 0,C 180,E1 -4509.138,E2 -4509.138} C_VEL
LIN {X 0,Y 531.045,Z 334.954,A -85,B 0,C 180,E1 -4512.225,E2 -4512.225} C_VEL
LIN {X 0,Y 531,Z 334.967,A -85,B 0,C 180,E1 -4515.35,E2 -4515.35} C_VEL
LIN {X 0,Y 530.994,Z 334.964,A -85,B 0,C 180,E1 -4518.521,E2 -4518.521} C_VEL
LIN {X 0,Y 531.003,Z 334.96,A -85,B 0,C 180,E1 -4520.938,E2 -4520.938} C_VEL
LIN {X 0,Y 530.969,Z 334.974,A -85,B 0,C 180,E1 -4524.225,E2 -4524.225} C_VEL
LIN {X 0,Y 531.006,Z 334.961,A -85,B 0,C 180,E1 -4526.744,E2 -4526.744} C_VEL
LIN {X 0,Y 530.985,Z 334.967,A -85,B 0,C 180,E1 -4529.323,E2 -4529.323} C_VEL
LIN {X 0,Y 530.969,Z 334.969,A -85,B 0,C 180,E1 -4532.1,E2 -4532.1} C_VEL
LIN {X 0,Y 530.987,Z 334.97,A -85,B 0,C 180,E1 -4534.853,E2 -4534.853} C_VEL
LIN {X 0,Y 530.971,Z 334.97,A -85,B 0,C 180,E1 -4537.507,E2 -4537.507} C_VEL
LIN {X 0,Y 530.987,Z 334.968,A -85,B 0,C 180,E1 -4540.433,E2 -4540.433} C_VEL
LIN {X 0,Y 530.968,Z 334.971,A -85,B 0,C 180,E1 -4543.494,E2 -4543.494} C_VEL
LIN {X 0,Y 530.965,Z 334.97,A -85,B 0,C 180,E1 -4543.56,E2 -4543.56} C_VEL
LIN {X 0,Y 530.294,Z 335.057,A -85,B 0,C 180,E1 -4544.194,E2 -4544.194} C_VEL
LIN {X 0,Y 527.45,Z 335.412,A -85,B 0,C 180,E1 -4545.223,E2 -4545.223} C_VEL
LIN {X 0,Y 525.046,Z 335.714,A -85,B 0,C 180,E1 -4546.051,E2 -4546.051} C_VEL
LIN {X 0,Y 524.008,Z 335.842,A -85,B 0,C 180,E1 -4546.691,E2 -4546.691} C_VEL
LIN {X 0,Y 523.921,Z 335.851,A -85,B 0,C 180,E1 -4546.907,E2 -4546.907} C_VEL
LIN {X 0,Y 523.83,Z 335.865,A -85,B 0,C 180,E1 -4548.897,E2 -4548.897} C_VEL
LIN {X 0,Y 523.77,Z 335.87,A -85,B 0,C 180,E1 -4549.904,E2 -4549.904} C_VEL
LIN {X 0,Y 523.694,Z 337.35,A -85,B 0,C 180,E1 -4551.879,E2 -4551.879} C_VEL
LIN {X 0,Y 523.674,Z 340.214,A -85,B 0,C 180,E1 -4554.95,E2 -4554.95} C_VEL
LIN {X 0,Y 523.624,Z 342.848,A -85,B 0,C 180,E1 -4557.734,E2 -4557.734} C_VEL
LIN {X 0,Y 523.555,Z 345.764,A -85,B 0,C 180,E1 -4560.755,E2 -4560.755} C_VEL
LIN {X 0,Y 523.493,Z 348.71,A -85,B 0,C 180,E1 -4563.702,E2 -4563.702} C_VEL
LIN {X 0,Y 523.48,Z 351.364,A -85,B 0,C 180,E1 -4566.248,E2 -4566.248} C_VEL
LIN {X 0,Y 523.413,Z 353.971,A -85,B 0,C 180,E1 -4568.744,E2 -4568.744} C_VEL
LIN {X 0,Y 523.42,Z 356.071,A -85,B 0,C 180,E1 -4570.724,E2 -4570.724} C_VEL
LIN {X 0,Y 527.441,Z 371.645,A -85,B 0,C 180,E1 -4571.209,E2 -4571.209} C_VEL
LIN {X 0,Y 527.139,Z 385.794,A -85,B 0,C 180,E1 -4571.632,E2 -4571.632} C_VEL
LIN {X 0,Y 526.719,Z 400.429,A -85,B 0,C 180,E1 -4572.228,E2 -4572.228} C_VEL
LIN {X 0,Y 526.258,Z 415.229,A -85,B 0,C 180,E1 -4573.014,E2 -4573.014} C_VEL
LIN {X 0,Y 525.766,Z 428.571,A -85,B 0,C 180,E1 -4573.897,E2 -4573.897} C_VEL
LIN {X 0,Y 525.193,Z 441.854,A -85,B 0,C 180,E1 -4574.973,E2 -4574.973} C_VEL
LIN {X 0,Y 524.779,Z 452.923,A -85,B 0,C 180,E1 -4576.05,E2 -4576.05} C_VEL
LIN {X 0,Y 524.394,Z 463.069,A -85,B 0,C 180,E1 -4577.224,E2 -4577.224} C_VEL
LIN {X 0,Y 524.053,Z 473.054,A -85,B 0,C 180,E1 -4578.591,E2 -4578.591} C_VEL
LIN {X 0,Y 523.783,Z 481.383,A -85,B 0,C 180,E1 -4579.954,E2 -4579.954} C_VEL
LIN {X 0,Y 523.614,Z 489.208,A -85,B 0,C 180,E1 -4581.509,E2 -4581.509} C_VEL
LIN {X 0,Y 523.483,Z 495.443,A -85,B 0,C 180,E1 -4583.06,E2 -4583.06} C_VEL
LIN {X 0,Y 523.441,Z 500.262,A -85,B 0,C 180,E1 -4584.607,E2 -4584.607} C_VEL
LIN {X 0,Y 523.402,Z 503.797,A -85,B 0,C 180,E1 -4586.15,E2 -4586.15} C_VEL
LIN {X 0,Y 523.333,Z 506.138,A -85,B 0,C 180,E1 -4587.691,E2 -4587.691} C_VEL
LIN {X 0,Y 523.246,Z 507.337,A -85,B 0,C 180,E1 -4589.23,E2 -4589.23} C_VEL
LIN {X 0,Y 523.247,Z 507.357,A -85,B 0,C 180,E1 -4590.769,E2 -4590.769} C_VEL
LIN {X 0,Y 523.333,Z 506.236,A -85,B 0,C 180,E1 -4592.309,E2 -4592.309} C_VEL
LIN {X 0,Y 523.402,Z 503.972,A -85,B 0,C 180,E1 -4593.849,E2 -4593.849} C_VEL
LIN {X 0,Y 523.438,Z 500.511,A -85,B 0,C 180,E1 -4595.393,E2 -4595.393} C_VEL
LIN {X 0,Y 523.481,Z 495.772,A -85,B 0,C 180,E1 -4596.94,E2 -4596.94} C_VEL
LIN {X 0,Y 523.612,Z 489.634,A -85,B 0,C 180,E1 -4598.49,E2 -4598.49} C_VEL
LIN {X 0,Y 523.775,Z 481.907,A -85,B 0,C 180,E1 -4600.045,E2 -4600.045} C_VEL
LIN {X 0,Y 524.002,Z 473.669,A -85,B 0,C 180,E1 -4601.41,E2 -4601.41} C_VEL
LIN {X 0,Y 524.365,Z 463.799,A -85,B 0,C 180,E1 -4602.776,E2 -4602.776} C_VEL
LIN {X 0,Y 524.748,Z 453.737,A -85,B 0,C 180,E1 -4603.95,E2 -4603.95} C_VEL
LIN {X 0,Y 525.191,Z 441.91,A -85,B 0,C 180,E1 -4605.111,E2 -4605.111} C_VEL
LIN {X 0,Y 525.773,Z 428.575,A -85,B 0,C 180,E1 -4606.192,E2 -4606.192} C_VEL
LIN {X 0,Y 526.278,Z 415.089,A -85,B 0,C 180,E1 -4607.085,E2 -4607.085} C_VEL
LIN {X 0,Y 526.721,Z 401.245,A -85,B 0,C 180,E1 -4607.821,E2 -4607.821} C_VEL
LIN {X 0,Y 527.083,Z 386.701,A -85,B 0,C 180,E1 -4608.425,E2 -4608.425} C_VEL
LIN {X 0,Y 527.403,Z 371.258,A -85,B 0,C 180,E1 -4608.893,E2 -4608.893} C_VEL
LIN {X 0,Y 523.414,Z 356.053,A -85,B 0,C 180,E1 -4609.357,E2 -4609.357} C_VEL
LIN {X 0,Y 523.435,Z 353.16,A -85,B 0,C 180,E1 -4612.113,E2 -4612.113} C_VEL
LIN {X 0,Y 523.444,Z 350.591,A -85,B 0,C 180,E1 -4614.596,E2 -4614.596} C_VEL
LIN {X 0,Y 523.51,Z 347.942,A -85,B 0,C 180,E1 -4617.157,E2 -4617.157} C_VEL
LIN {X 0,Y 523.545,Z 345.341,A -85,B 0,C 180,E1 -4619.78,E2 -4619.78} C_VEL
LIN {X 0,Y 523.62,Z 342.742,A -85,B 0,C 180,E1 -4622.471,E2 -4622.471} C_VEL
LIN {X 0,Y 523.668,Z 340.115,A -85,B 0,C 180,E1 -4625.246,E2 -4625.246} C_VEL
LIN {X 0,Y 523.696,Z 337.439,A -85,B 0,C 180,E1 -4628.12,E2 -4628.12} C_VEL
LIN {X 0,Y 523.771,Z 335.87,A -85,B 0,C 180,E1 -4630.108,E2 -4630.108} C_VEL
LIN {X 0,Y 523.928,Z 335.845,A -85,B 0,C 180,E1 -4632.458,E2 -4632.458} C_VEL
LIN {X 0,Y 523.955,Z 335.843,A -85,B 0,C 180,E1 -4635.308,E2 -4635.308} C_VEL
LIN {X 0,Y 523.96,Z 335.843,A -85,B 0,C 180,E1 -4638.689,E2 -4638.689} C_VEL
LIN {X 0,Y 523.917,Z 335.85,A -85,B 0,C 180,E1 -4641.898,E2 -4641.898} C_VEL
LIN {X 0,Y 523.938,Z 335.847,A -85,B 0,C 180,E1 -4644.908,E2 -4644.908} C_VEL
LIN {X 0,Y 523.939,Z 335.842,A -85,B 0,C 180,E1 -4647.679,E2 -4647.679} C_VEL
LIN {X 0,Y 523.969,Z 335.841,A -85,B 0,C 180,E1 -4650.673,E2 -4650.673} C_VEL
LIN {X 0,Y 523.977,Z 335.836,A -85,B 0,C 180,E1 -4653.729,E2 -4653.729} C_VEL
LIN {X 0,Y 523.935,Z 335.846,A -85,B 0,C 180,E1 -4656.271,E2 -4656.271} C_VEL
LIN {X 0,Y 523.945,Z 335.844,A -85,B 0,C 180,E1 -4658.767,E2 -4658.767} C_VEL
LIN {X 0,Y 523.953,Z 335.841,A -85,B 0,C 180,E1 -4661.221,E2 -4661.221} C_VEL
LIN {X 0,Y 523.94,Z 335.847,A -85,B 0,C 180,E1 -4663.639,E2 -4663.639} C_VEL
LIN {X 0,Y 523.939,Z 335.841,A -85,B 0,C 180,E1 -4666.028,E2 -4666.028} C_VEL
LIN {X 0,Y 524.013,Z 335.835,A -85,B 0,C 180,E1 -4668.394,E2 -4668.394} C_VEL
LIN {X 0,Y 524.004,Z 335.837,A -85,B 0,C 180,E1 -4671.516,E2 -4671.516} C_VEL
LIN {X 0,Y 524.083,Z 335.828,A -85,B 0,C 180,E1 -4674.614,E2 -4674.614} C_VEL
LIN {X 0,Y 524.11,Z 335.824,A -85,B 0,C 180,E1 -4677.694,E2 -4677.694} C_VEL
LIN {X 0,Y 524.123,Z 335.823,A -85,B 0,C 180,E1 -4680.768,E2 -4680.768} C_VEL
LIN {X 0,Y 524.073,Z 335.831,A -85,B 0,C 180,E1 -4683.075,E2 -4683.075} C_VEL
LIN {X 0,Y 524.045,Z 335.836,A -85,B 0,C 180,E1 -4686.159,E2 -4686.159} C_VEL
LIN {X 0,Y 523.997,Z 335.842,A -85,B 0,C 180,E1 -4689.262,E2 -4689.262} C_VEL
LIN {X 0,Y 524.007,Z 335.836,A -85,B 0,C 180,E1 -4691.743,E2 -4691.743} C_VEL
LIN {X 0,Y 523.991,Z 335.839,A -85,B 0,C 180,E1 -4695.052,E2 -4695.052} C_VEL
LIN {X 0,Y 523.962,Z 335.842,A -85,B 0,C 180,E1 -4697.969,E2 -4697.969} C_VEL
LIN {X 0,Y 523.97,Z 335.842,A -85,B 0,C 180,E1 -4700.41,E2 -4700.41} C_VEL
LIN {X 0,Y 523.915,Z 335.851,A -85,B 0,C 180,E1 -4702.893,E2 -4702.893} C_VEL
LIN {X 0,Y 523.951,Z 335.844,A -85,B 0,C 180,E1 -4705.419,E2 -4705.419} C_VEL
LIN {X 0,Y 523.968,Z 335.844,A -85,B 0,C 180,E1 -4707.999,E2 -4707.999} C_VEL
LIN {X 0,Y 523.951,Z 335.847,A -85,B 0,C 180,E1 -4710.856,E2 -4710.856} C_VEL
LIN {X 0,Y 523.959,Z 335.847,A -85,B 0,C 180,E1 -4713.735,E2 -4713.735} C_VEL
LIN {X 0,Y 523.921,Z 335.85,A -85,B 0,C 180,E1 -4716.405,E2 -4716.405} C_VEL
LIN {X 0,Y 523.922,Z 335.847,A -85,B 0,C 180,E1 -4719.085,E2 -4719.085} C_VEL
LIN {X 0,Y 523.955,Z 335.844,A -85,B 0,C 180,E1 -4722.119,E2 -4722.119} C_VEL
LIN {X 0,Y 523.972,Z 335.953,A -85,B 0,C 180,E1 -4725.369,E2 -4725.369} C_VEL
LIN {X 0,Y 524.773,Z 341.214,A -85,B 0,C 180,E1 -4727.963,E2 -4727.963} C_VEL
LIN {X 0,Y 524.944,Z 345.779,A -85,B 0,C 180,E1 -4730.012,E2 -4730.012} C_VEL
LIN {X 0,Y 524.709,Z 352.749,A -85,B 0,C 180,E1 -4732.935,E2 -4732.935} C_VEL
LIN {X 0,Y 524.511,Z 359.801,A -85,B 0,C 180,E1 -4735.753,E2 -4735.753} C_VEL
LIN {X 0,Y 524.361,Z 366.96,A -85,B 0,C 180,E1 -4738.486,E2 -4738.486} C_VEL
LIN {X 0,Y 524.23,Z 374.125,A -85,B 0,C 180,E1 -4741.143,E2 -4741.143} C_VEL
LIN {X 0,Y 524.064,Z 381.882,A -85,B 0,C 180,E1 -4743.963,E2 -4743.963} C_VEL
LIN {X 0,Y 523.895,Z 389.575,A -85,B 0,C 180,E1 -4746.688,E2 -4746.688} C_VEL
LIN {X 0,Y 523.807,Z 398.019,A -85,B 0,C 180,E1 -4749.584,E2 -4749.584} C_VEL
LIN {X 0,Y 523.784,Z 401.198,A -85,B 0,C 180,E1 -4750.655,E2 -4750.655} C_VEL
LIN {X 0,Y 527.455,Z 417.476,A -85,B 0,C 180,E1 -4751.09,E2 -4751.09} C_VEL
LIN {X 0,Y 527.148,Z 432.214,A -85,B 0,C 180,E1 -4751.501,E2 -4751.501} C_VEL
LIN {X 0,Y 526.786,Z 446.675,A -85,B 0,C 180,E1 -4752.056,E2 -4752.056} C_VEL
LIN {X 0,Y 526.34,Z 460.103,A -85,B 0,C 180,E1 -4752.717,E2 -4752.717} C_VEL
LIN {X 0,Y 525.822,Z 474.452,A -85,B 0,C 180,E1 -4753.6,E2 -4753.6} C_VEL
LIN {X 0,Y 525.404,Z 487.456,A -85,B 0,C 180,E1 -4754.583,E2 -4754.583} C_VEL
LIN {X 0,Y 524.91,Z 499.328,A -85,B 0,C 180,E1 -4755.659,E2 -4755.659} C_VEL
LIN {X 0,Y 524.51,Z 510.141,A -85,B 0,C 180,E1 -4756.834,E2 -4756.834} C_VEL
LIN {X 0,Y 524.154,Z 519.313,A -85,B 0,C 180,E1 -4758.006,E2 -4758.006} C_VEL
LIN {X 0,Y 523.943,Z 528.298,A -85,B 0,C 180,E1 -4759.372,E2 -4759.372} C_VEL
LIN {X 0,Y 523.699,Z 535.751,A -85,B 0,C 180,E1 -4760.733,E2 -4760.733} C_VEL
LIN {X 0,Y 523.534,Z 542.701,A -85,B 0,C 180,E1 -4762.286,E2 -4762.286} C_VEL
LIN {X 0,Y 523.44,Z 548.163,A -85,B 0,C 180,E1 -4763.834,E2 -4763.834} C_VEL
LIN {X 0,Y 523.322,Z 552.291,A -85,B 0,C 180,E1 -4765.379,E2 -4765.379} C_VEL
LIN {X 0,Y 523.358,Z 555.184,A -85,B 0,C 180,E1 -4766.921,E2 -4766.921} C_VEL
LIN {X 0,Y 523.272,Z 556.909,A -85,B 0,C 180,E1 -4768.461,E2 -4768.461} C_VEL
LIN {X 0,Y 523.243,Z 557.5,A -85,B 0,C 180,E1 -4770,E2 -4770} C_VEL
LIN {X 0,Y 523.272,Z 556.907,A -85,B 0,C 180,E1 -4771.54,E2 -4771.54} C_VEL
LIN {X 0,Y 523.358,Z 555.179,A -85,B 0,C 180,E1 -4773.079,E2 -4773.079} C_VEL
LIN {X 0,Y 523.323,Z 552.287,A -85,B 0,C 180,E1 -4774.622,E2 -4774.622} C_VEL
LIN {X 0,Y 523.451,Z 548.164,A -85,B 0,C 180,E1 -4776.166,E2 -4776.166} C_VEL
LIN {X 0,Y 523.535,Z 542.699,A -85,B 0,C 180,E1 -4777.715,E2 -4777.715} C_VEL
LIN {X 0,Y 523.699,Z 535.742,A -85,B 0,C 180,E1 -4779.268,E2 -4779.268} C_VEL
LIN {X 0,Y 523.988,Z 527.078,A -85,B 0,C 180,E1 -4780.823,E2 -4780.823} C_VEL
LIN {X 0,Y 524.233,Z 517.844,A -85,B 0,C 180,E1 -4782.194,E2 -4782.194} C_VEL
LIN {X 0,Y 524.599,Z 508.505,A -85,B 0,C 180,E1 -4783.362,E2 -4783.362} C_VEL
LIN {X 0,Y 525.011,Z 496.356,A -85,B 0,C 180,E1 -4784.636,E2 -4784.636} C_VEL
LIN {X 0,Y 525.483,Z 484.731,A -85,B 0,C 180,E1 -4785.645,E2 -4785.645} C_VEL
LIN {X 0,Y 525.966,Z 471.573,A -85,B 0,C 180,E1 -4786.596,E2 -4786.596} C_VEL
LIN {X 0,Y 526.386,Z 458.306,A -85,B 0,C 180,E1 -4787.382,E2 -4787.382} C_VEL
LIN {X 0,Y 526.883,Z 443.305,A -85,B 0,C 180,E1 -4788.09,E2 -4788.09} C_VEL
LIN {X 0,Y 527.22,Z 428.437,A -85,B 0,C 180,E1 -4788.621,E2 -4788.621} C_VEL
LIN {X 0,Y 527.344,Z 416.578,A -85,B 0,C 180,E1 -4788.934,E2 -4788.934} C_VEL
LIN {X 0,Y 523.788,Z 401.18,A -85,B 0,C 180,E1 -4789.351,E2 -4789.351} C_VEL
LIN {X 0,Y 523.881,Z 392.668,A -85,B 0,C 180,E1 -4792.233,E2 -4792.233} C_VEL
LIN {X 0,Y 524.04,Z 383.629,A -85,B 0,C 180,E1 -4795.414,E2 -4795.414} C_VEL
LIN {X 0,Y 524.214,Z 375.274,A -85,B 0,C 180,E1 -4798.421,E2 -4798.421} C_VEL
LIN {X 0,Y 524.319,Z 368.51,A -85,B 0,C 180,E1 -4800.923,E2 -4800.923} C_VEL
LIN {X 0,Y 524.479,Z 360.893,A -85,B 0,C 180,E1 -4803.819,E2 -4803.819} C_VEL
LIN {X 0,Y 524.672,Z 354.057,A -85,B 0,C 180,E1 -4806.515,E2 -4806.515} C_VEL
LIN {X 0,Y 524.857,Z 346.891,A -85,B 0,C 180,E1 -4809.497,E2 -4809.497} C_VEL
LIN {X 0,Y 524.906,Z 342.511,A -85,B 0,C 180,E1 -4811.428,E2 -4811.428} C_VEL
LIN {X 0,Y 524.31,Z 337.912,A -85,B 0,C 180,E1 -4813.628,E2 -4813.628} C_VEL
LIN {X 0,Y 523.958,Z 335.844,A -85,B 0,C 180,E1 -4814.692,E2 -4814.692} C_VEL
LIN {X 0,Y 523.953,Z 335.845,A -85,B 0,C 180,E1 -4817.881,E2 -4817.881} C_VEL
LIN {X 0,Y 523.924,Z 335.849,A -85,B 0,C 180,E1 -4820.916,E2 -4820.916} C_VEL
LIN {X 0,Y 523.931,Z 335.849,A -85,B 0,C 180,E1 -4823.828,E2 -4823.828} C_VEL
LIN {X 0,Y 523.944,Z 335.847,A -85,B 0,C 180,E1 -4826.636,E2 -4826.636} C_VEL
LIN {X 0,Y 523.958,Z 335.846,A -85,B 0,C 180,E1 -4829.356,E2 -4829.356} C_VEL
LIN {X 0,Y 523.981,Z 335.844,A -85,B 0,C 180,E1 -4832.281,E2 -4832.281} C_VEL
LIN {X 0,Y 523.955,Z 335.843,A -85,B 0,C 180,E1 -4834.582,E2 -4834.582} C_VEL
LIN {X 0,Y 523.913,Z 335.852,A -85,B 0,C 180,E1 -4837.107,E2 -4837.107} C_VEL
LIN {X 0,Y 523.982,Z 335.843,A -85,B 0,C 180,E1 -4839.866,E2 -4839.866} C_VEL
LIN {X 0,Y 523.97,Z 335.844,A -85,B 0,C 180,E1 -4842.837,E2 -4842.837} C_VEL
LIN {X 0,Y 523.981,Z 335.841,A -85,B 0,C 180,E1 -4845.236,E2 -4845.236} C_VEL
LIN {X 0,Y 524.016,Z 335.836,A -85,B 0,C 180,E1 -4848.394,E2 -4848.394} C_VEL
LIN {X 0,Y 524.007,Z 335.837,A -85,B 0,C 180,E1 -4851.516,E2 -4851.516} C_VEL
LIN {X 0,Y 524.086,Z 335.827,A -85,B 0,C 180,E1 -4854.614,E2 -4854.614} C_VEL
LIN {X 0,Y 524.115,Z 335.823,A -85,B 0,C 180,E1 -4857.695,E2 -4857.695} C_VEL
LIN {X 0,Y 524.128,Z 335.821,A -85,B 0,C 180,E1 -4860.768,E2 -4860.768} C_VEL
LIN {X 0,Y 524.077,Z 335.829,A -85,B 0,C 180,E1 -4863.075,E2 -4863.075} C_VEL
LIN {X 0,Y 524.052,Z 335.832,A -85,B 0,C 180,E1 -4866.159,E2 -4866.159} C_VEL
LIN {X 0,Y 524.003,Z 335.838,A -85,B 0,C 180,E1 -4869.262,E2 -4869.262} C_VEL
LIN {X 0,Y 524.007,Z 335.835,A -85,B 0,C 180,E1 -4871.739,E2 -4871.739} C_VEL
LIN {X 0,Y 523.997,Z 335.84,A -85,B 0,C 180,E1 -4875.052,E2 -4875.052} C_VEL
LIN {X 0,Y 523.968,Z 335.845,A -85,B 0,C 180,E1 -4877.969,E2 -4877.969} C_VEL
LIN {X 0,Y 523.976,Z 335.832,A -85,B 0,C 180,E1 -4880.41,E2 -4880.41} C_VEL
LIN {X 0,Y 523.914,Z 335.85,A -85,B 0,C 180,E1 -4882.894,E2 -4882.894} C_VEL
LIN {X 0,Y 523.988,Z 335.837,A -85,B 0,C 180,E1 -4886.02,E2 -4886.02} C_VEL
LIN {X 0,Y 523.943,Z 335.848,A -85,B 0,C 180,E1 -4888.875,E2 -4888.875} C_VEL
LIN {X 0,Y 523.924,Z 335.849,A -85,B 0,C 180,E1 -4891.544,E2 -4891.544} C_VEL
LIN {X 0,Y 523.944,Z 335.841,A -85,B 0,C 180,E1 -4894.289,E2 -4894.289} C_VEL
LIN {X 0,Y 523.916,Z 335.848,A -85,B 0,C 180,E1 -4897.132,E2 -4897.132} C_VEL
LIN {X 0,Y 523.94,Z 335.845,A -85,B 0,C 180,E1 -4900.13,E2 -4900.13} C_VEL
LIN {X 0,Y 523.939,Z 335.851,A -85,B 0,C 180,E1 -4902.459,E2 -4902.459} C_VEL
LIN {X 0,Y 523.959,Z 335.846,A -85,B 0,C 180,E1 -4905.309,E2 -4905.309} C_VEL
LIN {X 0,Y 523.921,Z 335.851,A -85,B 0,C 180,E1 -4906.907,E2 -4906.907} C_VEL
LIN {X 0,Y 523.232,Z 335.958,A -85,B 0,C 180,E1 -4907.549,E2 -4907.549} C_VEL
LIN {X 0,Y 520.319,Z 336.302,A -85,B 0,C 180,E1 -4908.589,E2 -4908.589} C_VEL
LIN {X 0,Y 517.849,Z 336.609,A -85,B 0,C 180,E1 -4909.427,E2 -4909.427} C_VEL
LIN {X 0,Y 516.77,Z 336.742,A -85,B 0,C 180,E1 -4910.073,E2 -4910.073} C_VEL
LIN {X 0,Y 516.672,Z 336.776,A -85,B 0,C 180,E1 -4910.292,E2 -4910.292} C_VEL
LIN {X 0,Y 516.634,Z 339.472,A -85,B 0,C 180,E1 -4913.38,E2 -4913.38} C_VEL
LIN {X 0,Y 516.582,Z 341.994,A -85,B 0,C 180,E1 -4916.096,E2 -4916.096} C_VEL
LIN {X 0,Y 516.529,Z 344.734,A -85,B 0,C 180,E1 -4919.003,E2 -4919.003} C_VEL
LIN {X 0,Y 516.455,Z 347.808,A -85,B 0,C 180,E1 -4922.194,E2 -4922.194} C_VEL
LIN {X 0,Y 516.393,Z 350.706,A -85,B 0,C 180,E1 -4925.045,E2 -4925.045} C_VEL
LIN {X 0,Y 516.369,Z 353.525,A -85,B 0,C 180,E1 -4927.745,E2 -4927.745} C_VEL
LIN {X 0,Y 516.332,Z 356.448,A -85,B 0,C 180,E1 -4930.456,E2 -4930.456} C_VEL
LIN {X 0,Y 520.498,Z 371.698,A -85,B 0,C 180,E1 -4930.939,E2 -4930.939} C_VEL
LIN {X 0,Y 520.577,Z 377.912,A -85,B 0,C 180,E1 -4931.117,E2 -4931.117} C_VEL
LIN {X 0,Y 520.239,Z 393.282,A -85,B 0,C 180,E1 -4931.66,E2 -4931.66} C_VEL
